END_VAR
// calculate Hour
	arCalculateEnergy_1H[LV01]( lrAccumulator := pmDev.DB07_01_5500.Basic.RealEnergy_IntoLoad);
	arCalculateEnergy_1H[DB_PR1_1]( lrAccumulator := pmDev.DB06_06_5500.Basic.RealEnergy_IntoLoad);
	arCalculateEnergy_1H[DB1]( lrAccumulator := pmDev.DB05_10_5500.Basic.RealEnergy_IntoLoad);
	arCalculateEnergy_1H[DB2]( lrAccumulator := pmDev.DB04_06_5500.Basic.RealEnergy_IntoLoad);
	arCalculateEnergy_1H[DB3]( lrAccumulator := pmDev.DB04_04_5500.Basic.RealEnergy_IntoLoad);
	arCalculateEnergy_1H[DB4]( lrAccumulator := pmDev.DB04_02_5500.Basic.RealEnergy_IntoLoad);
	arCalculateEnergy_1H[DB1_1]( lrAccumulator := pmDev.DB05_09_5350.Basic.RealEnergy_IntoLoad);
	arCalculateEnergy_1H[DB2_1]( lrAccumulator := pmDev.DB04_05_5350.Basic.RealEnergy_IntoLoad);
	arCalculateEnergy_1H[DB3_1]( lrAccumulator := pmDev.DB04_03_5350.Basic.RealEnergy_IntoLoad);
	arCalculateEnergy_1H[DB4_1]( lrAccumulator := pmDev.DB04_01_5350.Basic.RealEnergy_IntoLoad);
	arCalculateEnergy_1H[DB5]( lrAccumulator := pmDev.DB03_04_5500.Basic.RealEnergy_IntoLoad);
	arCalculateEnergy_1H[DB6]( lrAccumulator := pmDev.DB03_06_5500.Basic.RealEnergy_IntoLoad);
	arCalculateEnergy_1H[DB7]( lrAccumulator := pmDev.DB03_02_5500.Basic.RealEnergy_IntoLoad);
	arCalculateEnergy_1H[DB_MR]( lrAccumulator := pmDev.DB06_11_5500.Basic.RealEnergy_IntoLoad);
	arCalculateEnergy_1H[DB5_1]( lrAccumulator := pmDev.DB03_03_5350.Basic.RealEnergy_IntoLoad);
	arCalculateEnergy_1H[DB6_1]( lrAccumulator := pmDev.DB03_05_5350.Basic.RealEnergy_IntoLoad);
	arCalculateEnergy_1H[DB7_1]( lrAccumulator := pmDev.DB03_01_5350.Basic.RealEnergy_IntoLoad);
	arCalculateEnergy_1H[LV02]( lrAccumulator := pmDev.DB07_02_5500.Basic.RealEnergy_IntoLoad);
	arCalculateEnergy_1H[DB_PR1_2]( lrAccumulator := pmDev.DB06_05_5500.Basic.RealEnergy_IntoLoad);
	arCalculateEnergy_1H[DB_AIRCOMP]( lrAccumulator := pmDev.DB07_03_5500.Basic.RealEnergy_IntoLoad);
	arCalculateEnergy_1H[DB_AHU]( lrAccumulator := pmDev.DB06_07_5500.Basic.RealEnergy_IntoLoad);
	arCalculateEnergy_1H[DB8]( lrAccumulator := pmDev.DB05_04_5500.Basic.RealEnergy_IntoLoad);
	arCalculateEnergy_1H[DB9]( lrAccumulator := pmDev.DB05_06_5500.Basic.RealEnergy_IntoLoad);
	arCalculateEnergy_1H[DB10]( lrAccumulator := pmDev.DB05_08_5500.Basic.RealEnergy_IntoLoad);
	arCalculateEnergy_1H[DB8_1]( lrAccumulator := pmDev.DB05_03_5350.Basic.RealEnergy_IntoLoad);
	arCalculateEnergy_1H[DB9_1]( lrAccumulator := pmDev.DB05_05_5350.Basic.RealEnergy_IntoLoad);
	arCalculateEnergy_1H[DB10_1]( lrAccumulator := pmDev.DB05_07_5350.Basic.RealEnergy_IntoLoad);
	arCalculateEnergy_1H[A1]( lrAccumulator := pmDev.DB07_06_5350.Basic.RealEnergy_IntoLoad);
	arCalculateEnergy_1H[A2]( lrAccumulator := pmDev.DB07_07_5350.Basic.RealEnergy_IntoLoad);
	arCalculateEnergy_1H[A3]( lrAccumulator := pmDev.DB07_08_5350.Basic.RealEnergy_IntoLoad);
	arCalculateEnergy_1H[A4]( lrAccumulator := pmDev.DB07_09_5350.Basic.RealEnergy_IntoLoad);
	arCalculateEnergy_1H[A5]( lrAccumulator := pmDev.DB07_10_5350.Basic.RealEnergy_IntoLoad);
	arCalculateEnergy_1H[LP_PR1A]( lrAccumulator := pmDev.DB05_01_5350.Basic.RealEnergy_IntoLoad);
	arCalculateEnergy_1H[LP_PR1B]( lrAccumulator := pmDev.DB05_02_5350.Basic.RealEnergy_IntoLoad);
	arCalculateEnergy_1H[LP_PR2A]( lrAccumulator := pmDev.DB05_22_5350.Basic.RealEnergy_IntoLoad);
	arCalculateEnergy_1H[LP_PR2B]( lrAccumulator := pmDev.DB05_21_5350.Basic.RealEnergy_IntoLoad);
	arCalculateEnergy_1H[LP_PR3A]( lrAccumulator := pmDev.DB03_08_5350.Basic.RealEnergy_IntoLoad);
	arCalculateEnergy_1H[DB_WH]( lrAccumulator := pmDev.DB01_18_5500.Basic.RealEnergy_IntoLoad);
	arCalculateEnergy_1H[LP_PR3B]( lrAccumulator := pmDev.DB03_07_5350.Basic.RealEnergy_IntoLoad);
	arCalculateEnergy_1H[LP_PR4A]( lrAccumulator := pmDev.DB04_08_5350.Basic.RealEnergy_IntoLoad);
	arCalculateEnergy_1H[LP_PR4B]( lrAccumulator := pmDev.DB04_07_5350.Basic.RealEnergy_IntoLoad);
	arCalculateEnergy_1H[LP_BM]( lrAccumulator := pmDev.DB01_20_5500.Basic.RealEnergy_IntoLoad);
	arCalculateEnergy_1H[DB_BM]( lrAccumulator := pmDev.DB01_22_5500.Basic.RealEnergy_IntoLoad);
	arCalculateEnergy_1H[LV03]( lrAccumulator := pmDev.DB06_04_5500.Basic.RealEnergy_IntoLoad);
	arCalculateEnergy_1H[DB_MVAC1]( lrAccumulator := pmDev.DB07_05_5500.Basic.RealEnergy_IntoLoad);
	arCalculateEnergy_1H[DB_MVAC2]( lrAccumulator := pmDev.DB07_04_5500.Basic.RealEnergy_IntoLoad);
	arCalculateEnergy_1H[DB_OFF2]( lrAccumulator := pmDev.DB06_38_5500.Basic.RealEnergy_IntoLoad);
	arCalculateEnergy_1H[LP_EL1]( lrAccumulator := pmDev.DB06_03_5500.Basic.RealEnergy_IntoLoad);
	arCalculateEnergy_1H[LP_EL2]( lrAccumulator := pmDev.DB06_01_5500.Basic.RealEnergy_IntoLoad);
	arCalculateEnergy_1H[DB_OFF1]( lrAccumulator := pmDev.DB06_08_5500.Basic.RealEnergy_IntoLoad);
	arCalculateEnergy_1H[DB_KIT]( lrAccumulator := pmDev.DB06_33_5500.Basic.RealEnergy_IntoLoad);
	arCalculateEnergy_1H[LP_WH2]( lrAccumulator := pmDev.DB01_12_5350.Basic.RealEnergy_IntoLoad);
	arCalculateEnergy_1H[LP_WH1]( lrAccumulator := pmDev.DB01_11_5500.Basic.RealEnergy_IntoLoad);
	arCalculateEnergy_1H[CH4]( lrAccumulator := pmDev.DB07_11_5350.Basic.RealEnergy_IntoLoad);
	arCalculateEnergy_1H[CH5]( lrAccumulator := pmDev.DB07_12_5350.Basic.RealEnergy_IntoLoad);
	arCalculateEnergy_1H[CH6]( lrAccumulator := pmDev.DB07_13_5350.Basic.RealEnergy_IntoLoad);
	arCalculateEnergy_1H[LV04]( lrAccumulator := pmDev.DB06_02_5500.Basic.RealEnergy_IntoLoad);
	arCalculateEnergy_1H[DB_PR2]( lrAccumulator := pmDev.DB01_07_5500.Basic.RealEnergy_IntoLoad);
	arCalculateEnergy_1H[DB11]( lrAccumulator := pmDev.DB01_04_5500.Basic.RealEnergy_IntoLoad);
	arCalculateEnergy_1H[DB12]( lrAccumulator := pmDev.DB01_01_5500.Basic.RealEnergy_IntoLoad);
	arCalculateEnergy_1H[DB13]( lrAccumulator := pmDev.DB02_02_5500.Basic.RealEnergy_IntoLoad);
	arCalculateEnergy_1H[DB14]( lrAccumulator := pmDev.DB02_06_5500.Basic.RealEnergy_IntoLoad);
	arCalculateEnergy_1H[DB11_1]( lrAccumulator := pmDev.DB01_03_5350.Basic.RealEnergy_IntoLoad);
	arCalculateEnergy_1H[DB12_1]( lrAccumulator := pmDev.DB01_02_5350.Basic.RealEnergy_IntoLoad);
	arCalculateEnergy_1H[DB13_1]( lrAccumulator := pmDev.DB02_01_5350.Basic.RealEnergy_IntoLoad);
	arCalculateEnergy_1H[DB14_1]( lrAccumulator := pmDev.DB02_05_5350.Basic.RealEnergy_IntoLoad);
	arCalculateEnergy_1H[DB15]( lrAccumulator := pmDev.DB02_04_5500.Basic.RealEnergy_IntoLoad);
	arCalculateEnergy_1H[DB15_1]( lrAccumulator := pmDev.DB02_03_5350.Basic.RealEnergy_IntoLoad);
	arCalculateEnergy_1H[LP_PR5A]( lrAccumulator := pmDev.DB02_08_5350.Basic.RealEnergy_IntoLoad);
	arCalculateEnergy_1H[LP_PR5B]( lrAccumulator := pmDev.DB02_07_5350.Basic.RealEnergy_IntoLoad);
	arCalculateEnergy_1H[LP_PR6A]( lrAccumulator := pmDev.DB01_06_5350.Basic.RealEnergy_IntoLoad);
	arCalculateEnergy_1H[LP_PR6B]( lrAccumulator := pmDev.DB01_05_5350.Basic.RealEnergy_IntoLoad);
	arCalculateEnergy_1H[DB1_2]( lrAccumulator := pmDev.PowerMeter_DB1_2.Basic.RealEnergy_IntoLoad);
	arCalculateEnergy_1H[DB2_2]( lrAccumulator := pmDev.PowerMeter_DB2_2.Basic.RealEnergy_IntoLoad);
	arCalculateEnergy_1H[DB3_2]( lrAccumulator := pmDev.PowerMeter_DB3_2.Basic.RealEnergy_IntoLoad);
	arCalculateEnergy_1H[DB4_2]( lrAccumulator := pmDev.PowerMeter_DB4_2.Basic.RealEnergy_IntoLoad);
	arCalculateEnergy_1H[DB5_2]( lrAccumulator := pmDev.PowerMeter_DB5_2.Basic.RealEnergy_IntoLoad);
	arCalculateEnergy_1H[DB6_2]( lrAccumulator := pmDev.PowerMeter_DB6_2.Basic.RealEnergy_IntoLoad);
	arCalculateEnergy_1H[DB7_2]( lrAccumulator := pmDev.PowerMeter_DB7_2.Basic.RealEnergy_IntoLoad);
	arCalculateEnergy_1H[DB8_2]( lrAccumulator := pmDev.PowerMeter_DB8_2.Basic.RealEnergy_IntoLoad);
	arCalculateEnergy_1H[DB9_2]( lrAccumulator := pmDev.PowerMeter_DB9_2.Basic.RealEnergy_IntoLoad);
	arCalculateEnergy_1H[DB10_2]( lrAccumulator := pmDev.PowerMeter_DB10_2.Basic.RealEnergy_IntoLoad);
	arCalculateEnergy_1H[DB11_2]( lrAccumulator := pmDev.PowerMeter_DB11_2.Basic.RealEnergy_IntoLoad);
	arCalculateEnergy_1H[DB12_2]( lrAccumulator := pmDev.PowerMeter_DB12_2.Basic.RealEnergy_IntoLoad);
	arCalculateEnergy_1H[DB13_2]( lrAccumulator := pmDev.PowerMeter_DB13_2.Basic.RealEnergy_IntoLoad);
	arCalculateEnergy_1H[DB14_2]( lrAccumulator := pmDev.PowerMeter_DB14_2.Basic.RealEnergy_IntoLoad);
	arCalculateEnergy_1H[DB15_2]( lrAccumulator := pmDev.PowerMeter_DB15_2.Basic.RealEnergy_IntoLoad);
// calculate Day
	arCalculateEnergy_1D[LV01]( lrAccumulator := pmDev.DB07_01_5500.Basic.RealEnergy_IntoLoad);
	arCalculateEnergy_1D[DB_PR1_1]( lrAccumulator := pmDev.DB06_06_5500.Basic.RealEnergy_IntoLoad);
	arCalculateEnergy_1D[DB1]( lrAccumulator := pmDev.DB05_10_5500.Basic.RealEnergy_IntoLoad);
	arCalculateEnergy_1D[DB2]( lrAccumulator := pmDev.DB04_06_5500.Basic.RealEnergy_IntoLoad);
	arCalculateEnergy_1D[DB3]( lrAccumulator := pmDev.DB04_04_5500.Basic.RealEnergy_IntoLoad);
	arCalculateEnergy_1D[DB4]( lrAccumulator := pmDev.DB04_02_5500.Basic.RealEnergy_IntoLoad);
	arCalculateEnergy_1D[DB1_1]( lrAccumulator := pmDev.DB05_09_5350.Basic.RealEnergy_IntoLoad);
	arCalculateEnergy_1D[DB2_1]( lrAccumulator := pmDev.DB04_05_5350.Basic.RealEnergy_IntoLoad);
	arCalculateEnergy_1D[DB3_1]( lrAccumulator := pmDev.DB04_03_5350.Basic.RealEnergy_IntoLoad);
	arCalculateEnergy_1D[DB4_1]( lrAccumulator := pmDev.DB04_01_5350.Basic.RealEnergy_IntoLoad);
	arCalculateEnergy_1D[DB5]( lrAccumulator := pmDev.DB03_04_5500.Basic.RealEnergy_IntoLoad);
	arCalculateEnergy_1D[DB6]( lrAccumulator := pmDev.DB03_06_5500.Basic.RealEnergy_IntoLoad);
	arCalculateEnergy_1D[DB7]( lrAccumulator := pmDev.DB03_02_5500.Basic.RealEnergy_IntoLoad);
	arCalculateEnergy_1D[DB_MR]( lrAccumulator := pmDev.DB06_11_5500.Basic.RealEnergy_IntoLoad);
	arCalculateEnergy_1D[DB5_1]( lrAccumulator := pmDev.DB03_03_5350.Basic.RealEnergy_IntoLoad);
	arCalculateEnergy_1D[DB6_1]( lrAccumulator := pmDev.DB03_05_5350.Basic.RealEnergy_IntoLoad);
	arCalculateEnergy_1D[DB7_1]( lrAccumulator := pmDev.DB03_01_5350.Basic.RealEnergy_IntoLoad);
	arCalculateEnergy_1D[LV02]( lrAccumulator := pmDev.DB07_02_5500.Basic.RealEnergy_IntoLoad);
	arCalculateEnergy_1D[DB_PR1_2]( lrAccumulator := pmDev.DB06_05_5500.Basic.RealEnergy_IntoLoad);
	arCalculateEnergy_1D[DB_AIRCOMP]( lrAccumulator := pmDev.DB07_03_5500.Basic.RealEnergy_IntoLoad);
	arCalculateEnergy_1D[DB_AHU]( lrAccumulator := pmDev.DB06_07_5500.Basic.RealEnergy_IntoLoad);
	arCalculateEnergy_1D[DB8]( lrAccumulator := pmDev.DB05_04_5500.Basic.RealEnergy_IntoLoad);
	arCalculateEnergy_1D[DB9]( lrAccumulator := pmDev.DB05_06_5500.Basic.RealEnergy_IntoLoad);
	arCalculateEnergy_1D[DB10]( lrAccumulator := pmDev.DB05_08_5500.Basic.RealEnergy_IntoLoad);
	arCalculateEnergy_1D[DB8_1]( lrAccumulator := pmDev.DB05_03_5350.Basic.RealEnergy_IntoLoad);
	arCalculateEnergy_1D[DB9_1]( lrAccumulator := pmDev.DB05_05_5350.Basic.RealEnergy_IntoLoad);
	arCalculateEnergy_1D[DB10_1]( lrAccumulator := pmDev.DB05_07_5350.Basic.RealEnergy_IntoLoad);
	arCalculateEnergy_1D[A1]( lrAccumulator := pmDev.DB07_06_5350.Basic.RealEnergy_IntoLoad);
	arCalculateEnergy_1D[A2]( lrAccumulator := pmDev.DB07_07_5350.Basic.RealEnergy_IntoLoad);
	arCalculateEnergy_1D[A3]( lrAccumulator := pmDev.DB07_08_5350.Basic.RealEnergy_IntoLoad);
	arCalculateEnergy_1D[A4]( lrAccumulator := pmDev.DB07_09_5350.Basic.RealEnergy_IntoLoad);
	arCalculateEnergy_1D[A5]( lrAccumulator := pmDev.DB07_10_5350.Basic.RealEnergy_IntoLoad);
	arCalculateEnergy_1D[LP_PR1A]( lrAccumulator := pmDev.DB05_01_5350.Basic.RealEnergy_IntoLoad);
	arCalculateEnergy_1D[LP_PR1B]( lrAccumulator := pmDev.DB05_02_5350.Basic.RealEnergy_IntoLoad);
	arCalculateEnergy_1D[LP_PR2A]( lrAccumulator := pmDev.DB05_22_5350.Basic.RealEnergy_IntoLoad);
	arCalculateEnergy_1D[LP_PR2B]( lrAccumulator := pmDev.DB05_21_5350.Basic.RealEnergy_IntoLoad);
	arCalculateEnergy_1D[LP_PR3A]( lrAccumulator := pmDev.DB03_08_5350.Basic.RealEnergy_IntoLoad);
	arCalculateEnergy_1D[DB_WH]( lrAccumulator := pmDev.DB01_18_5500.Basic.RealEnergy_IntoLoad);
	arCalculateEnergy_1D[LP_PR3B]( lrAccumulator := pmDev.DB03_07_5350.Basic.RealEnergy_IntoLoad);
	arCalculateEnergy_1D[LP_PR4A]( lrAccumulator := pmDev.DB04_08_5350.Basic.RealEnergy_IntoLoad);
	arCalculateEnergy_1D[LP_PR4B]( lrAccumulator := pmDev.DB04_07_5350.Basic.RealEnergy_IntoLoad);
	arCalculateEnergy_1D[LP_BM]( lrAccumulator := pmDev.DB01_20_5500.Basic.RealEnergy_IntoLoad);
	arCalculateEnergy_1D[DB_BM]( lrAccumulator := pmDev.DB01_22_5500.Basic.RealEnergy_IntoLoad);
	arCalculateEnergy_1D[LV03]( lrAccumulator := pmDev.DB06_04_5500.Basic.RealEnergy_IntoLoad);
	arCalculateEnergy_1D[DB_MVAC1]( lrAccumulator := pmDev.DB07_05_5500.Basic.RealEnergy_IntoLoad);
	arCalculateEnergy_1D[DB_MVAC2]( lrAccumulator := pmDev.DB07_04_5500.Basic.RealEnergy_IntoLoad);
	arCalculateEnergy_1D[DB_OFF2]( lrAccumulator := pmDev.DB06_38_5500.Basic.RealEnergy_IntoLoad);
	arCalculateEnergy_1D[LP_EL1]( lrAccumulator := pmDev.DB06_03_5500.Basic.RealEnergy_IntoLoad);
	arCalculateEnergy_1D[LP_EL2]( lrAccumulator := pmDev.DB06_01_5500.Basic.RealEnergy_IntoLoad);
	arCalculateEnergy_1D[DB_OFF1]( lrAccumulator := pmDev.DB06_08_5500.Basic.RealEnergy_IntoLoad);
	arCalculateEnergy_1D[DB_KIT]( lrAccumulator := pmDev.DB06_33_5500.Basic.RealEnergy_IntoLoad);
	arCalculateEnergy_1D[LP_WH2]( lrAccumulator := pmDev.DB01_12_5350.Basic.RealEnergy_IntoLoad);
	arCalculateEnergy_1D[LP_WH1]( lrAccumulator := pmDev.DB01_11_5500.Basic.RealEnergy_IntoLoad);
	arCalculateEnergy_1D[CH4]( lrAccumulator := pmDev.DB07_11_5350.Basic.RealEnergy_IntoLoad);
	arCalculateEnergy_1D[CH5]( lrAccumulator := pmDev.DB07_12_5350.Basic.RealEnergy_IntoLoad);
	arCalculateEnergy_1D[CH6]( lrAccumulator := pmDev.DB07_13_5350.Basic.RealEnergy_IntoLoad);
	arCalculateEnergy_1D[LV04]( lrAccumulator := pmDev.DB06_02_5500.Basic.RealEnergy_IntoLoad);
	arCalculateEnergy_1D[DB_PR2]( lrAccumulator := pmDev.DB01_07_5500.Basic.RealEnergy_IntoLoad);
	arCalculateEnergy_1D[DB11]( lrAccumulator := pmDev.DB01_04_5500.Basic.RealEnergy_IntoLoad);
	arCalculateEnergy_1D[DB12]( lrAccumulator := pmDev.DB01_01_5500.Basic.RealEnergy_IntoLoad);
	arCalculateEnergy_1D[DB13]( lrAccumulator := pmDev.DB02_02_5500.Basic.RealEnergy_IntoLoad);
	arCalculateEnergy_1D[DB14]( lrAccumulator := pmDev.DB02_06_5500.Basic.RealEnergy_IntoLoad);
	arCalculateEnergy_1D[DB11_1]( lrAccumulator := pmDev.DB01_03_5350.Basic.RealEnergy_IntoLoad);
	arCalculateEnergy_1D[DB12_1]( lrAccumulator := pmDev.DB01_02_5350.Basic.RealEnergy_IntoLoad);
	arCalculateEnergy_1D[DB13_1]( lrAccumulator := pmDev.DB02_01_5350.Basic.RealEnergy_IntoLoad);
	arCalculateEnergy_1D[DB14_1]( lrAccumulator := pmDev.DB02_05_5350.Basic.RealEnergy_IntoLoad);
	arCalculateEnergy_1D[DB15]( lrAccumulator := pmDev.DB02_04_5500.Basic.RealEnergy_IntoLoad);
	arCalculateEnergy_1D[DB15_1]( lrAccumulator := pmDev.DB02_03_5350.Basic.RealEnergy_IntoLoad);
	arCalculateEnergy_1D[LP_PR5A]( lrAccumulator := pmDev.DB02_08_5350.Basic.RealEnergy_IntoLoad);
	arCalculateEnergy_1D[LP_PR5B]( lrAccumulator := pmDev.DB02_07_5350.Basic.RealEnergy_IntoLoad);
	arCalculateEnergy_1D[LP_PR6A]( lrAccumulator := pmDev.DB01_06_5350.Basic.RealEnergy_IntoLoad);
	arCalculateEnergy_1D[LP_PR6B]( lrAccumulator := pmDev.DB01_05_5350.Basic.RealEnergy_IntoLoad);
	arCalculateEnergy_1D[DB1_2]( lrAccumulator := pmDev.PowerMeter_DB1_2.Basic.RealEnergy_IntoLoad);
	arCalculateEnergy_1D[DB2_2]( lrAccumulator := pmDev.PowerMeter_DB2_2.Basic.RealEnergy_IntoLoad);
	arCalculateEnergy_1D[DB3_2]( lrAccumulator := pmDev.PowerMeter_DB3_2.Basic.RealEnergy_IntoLoad);
	arCalculateEnergy_1D[DB4_2]( lrAccumulator := pmDev.PowerMeter_DB4_2.Basic.RealEnergy_IntoLoad);
	arCalculateEnergy_1D[DB5_2]( lrAccumulator := pmDev.PowerMeter_DB5_2.Basic.RealEnergy_IntoLoad);
	arCalculateEnergy_1D[DB6_2]( lrAccumulator := pmDev.PowerMeter_DB6_2.Basic.RealEnergy_IntoLoad);
	arCalculateEnergy_1D[DB7_2]( lrAccumulator := pmDev.PowerMeter_DB7_2.Basic.RealEnergy_IntoLoad);
	arCalculateEnergy_1D[DB8_2]( lrAccumulator := pmDev.PowerMeter_DB8_2.Basic.RealEnergy_IntoLoad);
	arCalculateEnergy_1D[DB9_2]( lrAccumulator := pmDev.PowerMeter_DB9_2.Basic.RealEnergy_IntoLoad);
	arCalculateEnergy_1D[DB10_2]( lrAccumulator := pmDev.PowerMeter_DB10_2.Basic.RealEnergy_IntoLoad);
	arCalculateEnergy_1D[DB11_2]( lrAccumulator := pmDev.PowerMeter_DB11_2.Basic.RealEnergy_IntoLoad);
	arCalculateEnergy_1D[DB12_2]( lrAccumulator := pmDev.PowerMeter_DB12_2.Basic.RealEnergy_IntoLoad);
	arCalculateEnergy_1D[DB13_2]( lrAccumulator := pmDev.PowerMeter_DB13_2.Basic.RealEnergy_IntoLoad);
	arCalculateEnergy_1D[DB14_2]( lrAccumulator := pmDev.PowerMeter_DB14_2.Basic.RealEnergy_IntoLoad);
	arCalculateEnergy_1D[DB15_2]( lrAccumulator := pmDev.PowerMeter_DB15_2.Basic.RealEnergy_IntoLoad);
//FIFO Hour
	// // Check NEw Hour ( in the last Meter => it's mean all the calculate in 1 hour is updated)	
	IF arCalculateEnergy_1H[pmDev.numAllMeter-1].bNewPeriodAlarm THEN
		FIFOEnergyTimestruct_1H.MR_AddValue( Value := arCalculateEnergy_1H[pmDev.numAllMeter-1].previousTimestampOut);
		FOR iLoop := 0 TO pmDev.numAllMeter-1 DO
			arFIFOEnergy_1H[iLoop].MR_AddValue( Value := arCalculateEnergy_1H[iLoop].accumulatedValueOut);
			arCalculateEnergy_1H[iLoop].MR_Acknowledge();
		END_FOR
	END_IF	
// Check NEw Day ( in the last Meter => it's mean all the calculate in 1 day is updated)	
	IF arCalculateEnergy_1D[pmDev.numAllMeter-1].bNewPeriodAlarm THEN
		FIFOEnergyTimestruct_1D.MR_AddValue(  Value := arCalculateEnergy_1H[pmDev.numAllMeter-1].previousTimestampOut);
		FOR iLoop := 0 TO pmDev.numAllMeter-1 DO
			// round number before go to the FIFO
			arFIFOEnergy_1D[iLoop].MR_AddValue(
				Value := F_RoundLrealEx( 
					lrIn := arCalculateEnergy_1D[iLoop].accumulatedValueOut,
					iPrecision := 0)
			);
			// Ack The Calculate
			arCalculateEnergy_1D[iloop].MR_Acknowledge();
		END_FOR

	END_IF
	
CASE eStateReport OF
	STATE_REPORT_WAIT:
		// Check the last one FIFO[-1] hour if have data => request report to Aveva.
			IF arFIFOEnergy_1H[pmDev.numAllMeter-1].DataReady  THEN
				eStateReport := STATE_REPORT_ENERGY_HOUR_REQUEST;
		// Check the last one FIFO[-1] hour if have data => request report to Aveva.
			ELSIF arFIFOEnergy_1D[pmDev.numAllMeter-1].DataReady  THEN
				eStateReport := STATE_REPORT_ENERGY_DAY_REQUEST;
			END_IF;
			
	STATE_REPORT_ENERGY_HOUR_REQUEST:
		sDateAndTimeReportAveva := TimeStruct_To_sTimeAveva(timestruct := FIFOEnergyTimestruct_1H.OldestData, typeFormat := 5 );
		sMsReportAveva			:= WORD_TO_STRING ( FIFOEnergyTimestruct_1H.OldestData.wMilliseconds);
		
		fbMachineLogger.MR_AddLogs( sLogMessage :=  CONCAT('REPORT_ENERGY_HOUR_REQUEST  ', sDateAndTimeReportAveva  ));
		eStateReport := STATE_REPORT_ENERGY_HOUR_ACTIVE_REQUEST;
	
	STATE_REPORT_ENERGY_HOUR_ACTIVE_REQUEST	:
		tonPrepareValue( IN := TRUE,
							PT := tTimePrepareValue);
		IF tonPrepareValue.Q THEN
			tonPrepareValue( IN := FALSE);
			bEnergyReportHourEvent := TRUE;
			eStateReport := STATE_REPORT_ENERGY_HOUR_WAIT_ACK;
		END_IF
	
	STATE_REPORT_ENERGY_HOUR_WAIT_ACK:
		IF bEnergyReportHourEvent = FALSE THEN
			FOR iLoop := 0 TO pmDev.numAllMeter-1 DO
				arFIFOEnergy_1H[iLoop].MR_AckGetValue();
			END_FOR
			FIFOEnergyTimestruct_1H.MR_AckGetValue();
			fbMachineLogger.MR_AddLogs( sLogMessage :=  'REPORT_ENERGY_HOUR_ACKed  ');
			eStateReport := STATE_REPORT_WAIT;
		END_IF
				
	STATE_REPORT_ENERGY_DAY_REQUEST:
		CalculateVirtualObject();
		sDateAndTimeReportAveva := TimeStruct_To_sTimeAveva(timestruct := FIFOEnergyTimestruct_1D.OldestData, typeFormat := 5 );
	 	sMsReportAveva			:= WORD_TO_STRING ( FIFOEnergyTimestruct_1D.OldestData.wMilliseconds);
		bEnergyReportDayEvent := TRUE;
		fbMachineLogger.MR_AddLogs( sLogMessage :=  CONCAT('REPORT_ENERGY_DAY_REQUEST  ', sDateAndTimeReportAveva  ));
		eStateReport := STATE_REPORT_ENERGY_DAY_ACTIVE_REQUEST;
		
	STATE_REPORT_ENERGY_DAY_ACTIVE_REQUEST	:
		tonPrepareValue( IN := TRUE,
							PT := tTimePrepareValue);
		IF tonPrepareValue.Q THEN
			tonPrepareValue( IN := FALSE);
			bEnergyReportDayEvent := TRUE;
			eStateReport := STATE_REPORT_ENERGY_DAY_WAIT_ACK;
		END_IF	
		
	STATE_REPORT_ENERGY_DAY_WAIT_ACK:
		IF bEnergyReportDayEvent = FALSE THEN
			FOR iLoop := 0 TO pmDev.numAllMeter-1 DO
				arFIFOEnergy_1D[iLoop].MR_AckGetValue();	
			END_FOR

			FIFOEnergyTimestruct_1D.MR_AckGetValue();
			fbMachineLogger.MR_AddLogs( sLogMessage :=  'REPORT_ENERGY_HOUR_ACKed  ');
			eStateReport := STATE_REPORT_WAIT;
		END_IF
END_CASE
END_METHOD

END_PROGRAM

// ---- POUs/CalAccum/FB_CalCulateAccumulation.TcPOU
FUNCTION_BLOCK FB_CalCulateAccumulation
VAR_INPUT
	lrAccumulator : LREAL  := 0;
	
END_VAR
VAR_OUTPUT
	accumulatedValueOut : LREAL;// value = lrAccumulator(timeNew) - lrAccumulator(timeOld)
	previousTimestampOut	: TIMESTRUCT;// TimeOld
	bNewPeriodAlarm : BOOL;// Remain True in 30s if not be ackNowledge
	
END_VAR
VAR

	
	eCpHour		: E_CompareTime;
	eCpDay 		: E_CompareTime;
	eCpMonth	: E_CompareTime;
	eCpYear		: E_CompareTime;
	eCpMinute	: E_CompareTime;
	eSameTime : E_CompareTime;
	eNewTime : E_CompareTime;
	eRfTimeCompare : REFERENCE TO E_CompareTime;
	sName 		: STRING;
	eState : UINT;
	TonRemainOutput : TON;
	eTimeAccumulate : E_CompareTime;
	bInit : BOOL;
	bReset : BOOL;
	bRequestUpdate_ValueInLastTime: BOOL;
END_VAR

VAR PERSISTENT 
	bUpdatedValueLastHour : BOOL;// reject Power OFF unexpected
	previousTimestamp	: TIMESTRUCT;
	ValueInLastTime : LREAL;
	accumulatedValue : LREAL;
	
	
END_VAR
VAR CONSTANT
	eStateUinitialized : UINT := 0;
	eStateInit : UINT := 10;
	eStateRun : UINT := 20;
	eStateReset : UINT := 100;
	TimeNewPeriodAlarm : TIME := T#30s;
END_VAR



				
CASE eState OF
	eStateUinitialized: // unInitialized
		;// will go to eStateInit if MR_Run is called 
		
	eStateInit: 
		;// will call by MR_Init
		
	eStateRun: //StateRun
		MS_Run();
		
	eStateReset :
		MS_Reset();
	
END_CASE

IF eState > 0 AND bReset THEN
	eState := eStateReset;
END_IF

PROPERTY isInitDone : bool
GET
END_GET
END_PROPERTY

PROPERTY isRuning : bool
GET
isRuning := eState = eStateRun;
END_GET
END_PROPERTY

// if not return true , check the Current time and PreviousTime in fb
METHOD MR_Acknowledge : BOOL
VAR_INPUT
END_VAR
bNewPeriodAlarm := FALSE;
IF eRfTimeCompare = eSameTime THEN
	MR_Acknowledge := TRUE;
END_IF
END_METHOD

METHOD MR_Init : BOOL
VAR_INPUT
END_VAR

IF eState = eStateUinitialized THEN// init;
	bInit := true;
 
	IF MS_Init() THEN
		MR_Init := TRUE;
		eState := eStateRun;
	END_IF


END_IF
END_METHOD

METHOD MR_Reset : BOOL
VAR_INPUT
END_VAR
bReset := TRUE;
IF eState = eStateUinitialized THEN
	MR_Reset := TRUE;
	bReset := false;
END_IF
END_METHOD

METHOD Protected MS_Init : BOOL
VAR_INPUT
END_VAR
CASE eTimeAccumulate OF
	NEW_MINUTE :
		eSameTime := SAME_MINUTE;
		eNewTime := NEW_MINUTE;
		eRfTimeCompare REF= eCpMinute;
		MS_Init := TRUE;
	NEW_HOUR :
		eSameTime := SAME_HOUR;
		eNewTime := NEW_HOUR;
		eRfTimeCompare REF= eCpHour;
		MS_Init := TRUE;
	NEW_DAY	:
		eSameTime := SAME_DAY;
		eNewTime := NEW_DAY;
		eRfTimeCompare REF= eCpDay;
		MS_Init := TRUE;
	NEW_MONTH:
		eSameTime := SAME_MONTH;
		eNewTime := NEW_MONTH;
		eRfTimeCompare REF= eCpMonth;
		MS_Init := TRUE;
	NEW_YEAR:
		eSameTime := SAME_YEAR;
		eNewTime := NEW_YEAR;
		eRfTimeCompare REF= eCpYear;
		MS_Init := true;
END_CASE
END_METHOD

METHOD protected MS_Reset : BOOL
VAR_INPUT
END_VAR
//retainvalue
	
	bUpdatedValueLastHour := FALSE;
	previousTimestamp.wYear := 0;
	previousTimestamp.wMonth := 0;
	previousTimestamp.wDay := 0;
	previousTimestamp.wMinute := 0;
	previousTimestamp.wSecond := 0;
	previousTimestamp.wMilliseconds := 0;
	ValueInLastTime := 0 ;
	accumulatedValue := 0 ;
// out_put
	accumulatedValueOut := 0;
	previousTimestampOut.wYear := 0;
	previousTimestampOut.wMonth := 0;
	previousTimestampOut.wDay := 0;
	previousTimestampOut.wMinute := 0;
	previousTimestampOut.wSecond := 0;
	previousTimestampOut.wMilliseconds := 0;
	bNewPeriodAlarm := false;// Remain True 
	
// 	RETURN TO uninit
	eState := eStateUinitialized;
	eRfTimeCompare REF= 0;
END_METHOD

METHOD Protected MS_Run : BOOL
VAR_INPUT
END_VAR
	CompareTime(	timestruct1 := previousTimestamp,
					timestruct2 := GVL.fbMachineTime.systemTime,
					eCpMinute => eCpMinute, 
					eCpHour => eCpHour,
					eCpDay => eCpDay,
					eCpMonth => eCpMonth,
					ecpYear => eCpYear);

	IF eRfTimeCompare = eNewTime THEN
		// update to output
		accumulatedValueOut := accumulatedValue;
		previousTimestampOut := previousTimestamp;
		bNewPeriodAlarm := TRUE;
		// update the the last hour and time
		bUpdatedValueLastHour := FALSE;
		IF lrAccumulator > 0.1 THEN
			ValueInLastTime := lrAccumulator;
			bRequestUpdate_ValueInLastTime := FALSE;
			// UpdateOK
			bUpdatedValueLastHour := TRUE;
		ELSE
			bRequestUpdate_ValueInLastTime := TRUE;
		END_IF
		ValueInLastTime := lrAccumulator;
		previousTimestamp := GVL.fbMachineTime.systemTime;

	
	ELSIF eRfTimeCompare = eSameTime AND bUpdatedValueLastHour THEN
		IF lrAccumulator > 0.1 THEN // reject the situation that just TURN ON IPC so lrAccumulator = -8888888888888888.444444444444
			accumulatedValue := lrAccumulator - ValueInLastTime;
		END_IF
	ELSIF eRfTimeCompare = eSameTime AND NOT bUpdatedValueLastHour THEN
		ValueInLastTime := lrAccumulator;
		previousTimestamp := GVL.fbMachineTime.systemTime;
	ELSE
		; //invalid time Compare
	

	END_IF
	
TonRemainOutput( IN := bNewPeriodAlarm , PT := TimeNewPeriodAlarm);

IF TonRemainOutput.Q THEN
	bNewPeriodAlarm := false;
END_IF
IF bRequestUpdate_ValueInLastTime THEN
	IF lrAccumulator > 0.1 THEN
		ValueInLastTime := lrAccumulator;
		bRequestUpdate_ValueInLastTime := FALSE;
		// UpdateOK
		bUpdatedValueLastHour := TRUE;
	END_IF
END_IF
END_METHOD

PROPERTY Name : string
GET
Name := sName;
END_GET
SET
sName := Name;
END_SET
END_PROPERTY

// Set TimeAccumulate before call Mr_Init.
//NEW_MINUTE := 5,
//	NEW_HOUR := 10,
//	NEW_DAY	:= 20,
//	NEW_MONTH := 30,
//	NEW_YEAR	:= 32,
PROPERTY TimeAccumulate : E_CompareTime
GET
TimeAccumulate := eTimeAccumulate;
END_GET
SET
eTimeAccumulate := TimeAccumulate;
END_SET
END_PROPERTY

END_FUNCTION_BLOCK

// ---- Function/CompareTime.TcPOU
FUNCTION CompareTime : E_CompareTime
VAR_INPUT
		timestruct1 : TIMESTRUCT;//TIMEPREVIOUS
		timestruct2 : TIMESTRUCT;// TIME NOW
END_VAR
VAR_OUTPUT
	eCpMinute	: E_CompareTime;
	eCpHour		: E_CompareTime;
	eCpDay		: E_CompareTime;
	eCpMonth	: E_CompareTime;
	ecpYear		: E_CompareTime;
END_VAR

IF timestruct1.wYear < timestruct2.wYear THEN
	CompareTime := NEW_YEAR;
	ecpYear := NEW_YEAR;
	eCpMonth := NEW_MONTH;
	eCpDay := NEW_DAY;
	eCpHour := NEW_HOUR;
	eCpMinute := NEW_MINUTE;
ELSIF timestruct1.wYear > timestruct2.wYear THEN
		CompareTime := INVALID_PRE_TIME;
ELSE 
	ecpYear := SAME_YEAR;
	IF timestruct1.wMonth < timestruct2.wMonth THEN
		CompareTime := NEW_MONTH;
		eCpMonth := NEW_MONTH;
		eCpDay := NEW_DAY;
		eCpHour := NEW_HOUR;
		eCpMinute := NEW_MINUTE;
	ELSIF  timestruct1.wMonth > timestruct2.wMonth THEN
			CompareTime := INVALID_PRE_TIME;
	ELSE
		eCpMonth := SAME_MONTH;
		IF timestruct1.wDay < timestruct2.wDay THEN
			CompareTime := NEW_DAY;
			eCpDay := NEW_DAY;
			eCpHour := NEW_HOUR;
			eCpMinute := NEW_MINUTE;
		ELSIF timestruct1.wDay > timestruct2.wDay THEN
			CompareTime := INVALID_PRE_TIME;
		ELSE 
			eCpDay := SAME_DAY;
			IF timestruct1.wHour < timestruct2.wHour THEN
				CompareTime := NEW_HOUR;
				eCpHour := NEW_HOUR;
				eCpMinute := NEW_MINUTE;
			ELSIF timestruct1.wHour > timestruct2.wHour THEN
				CompareTime := INVALID_PRE_TIME; 
			ELSE
				eCpHour := SAME_HOUR;
				IF timestruct1.wMinute < timestruct2.wMinute THEN
					CompareTime := NEW_MINUTE;
					eCpMinute := NEW_MINUTE;
				ELSIF timestruct1.wMinute > timestruct2.wMinute THEN
					CompareTime := INVALID_PRE_TIME; 
				ELSE
					CompareTime := SAME_MINUTE;	
					eCpMinute := SAME_MINUTE;
			END_IF
			END_IF
		END_IF

	END_IF
END_IF

END_FUNCTION

// ---- POUs/FIFO/FB_FIFO_Lreal.TcPOU
FUNCTION_BLOCK FB_FIFO_Lreal EXTENDS FB_Universal_FIFO IMPLEMENTS I_FIFO_Lreal
VAR_INPUT
  
END_VAR

VAR
  
END_VAR

VAR_OUTPUT
	OldestData : LREAL;
END_VAR
VAR PERSISTENT
	Queue : ARRAY[0..MaxQueueSize-1] OF LREAL;  // FIFO queue (size is 100 elements)
END_VAR



//    // Log new data only if LogData is TRUE
//    IF rTrigLogData.Q THEN
//        IF Count < MaxQueueSize THEN
//            Queue[Head] := NewEnergyData;
//            Head := (Head + 1) MOD MaxQueueSize;
//            Count := Count + 1;
//        ELSE
//            // FIFO is full, overwrite old data if needed
//            Tail := (Tail + 1) MOD MaxQueueSize;
//            Queue[Head] := NewEnergyData;
//            Head := (Head + 1) MOD MaxQueueSize;
//            // Tail position is updated
//        END_IF
//        DataReady := TRUE;  // New data is now ready to be processed
     
//    END_IF

    // Retrieve and manage oldest data for processing

// if dataready return true, else return false
METHOD  MR_AckGetValue : BOOL
VAR_INPUT
END_VAR
SUPER^.MR_AckGetValue();
  OldestData := Queue[Tail];
 MR_AckGetValue := true;
END_METHOD

METHOD MR_AddValue : BOOL
VAR_INPUT
		Value : LREAL;
END_VAR
  IF Count < MaxQueueSize THEN
            Queue[Head] := Value;
            Head := (Head + 1) MOD MaxQueueSize;
            Count := Count + 1;
  ELSE
            // FIFO is full, overwrite old data if needed
            Tail := (Tail + 1) MOD MaxQueueSize;
            Queue[Head] := Value;
            Head := (Head + 1) MOD MaxQueueSize;
            // Tail position is updated
			
  END_IF
  
  OldestData := Queue[Tail];
  bDataReady := TRUE; 
  
  
  MR_AddValue := true;
END_METHOD

// need overide to reset oldestValue
METHOD MR_Reset : BOOL
VAR_INPUT
END_VAR
SUPER^.MR_Reset();
OldestData := 0;
MR_Reset := true;
END_METHOD

PROPERTY oOldestValue : Lreal
GET
oOldestValue := OldestData;
END_GET
END_PROPERTY

END_FUNCTION_BLOCK

// ---- POUs/FIFO/FB_Universal_FIFO.TcPOU
FUNCTION_BLOCK ABSTRACT FB_Universal_FIFO IMPLEMENTS I_Universal_FIFO

VAR PERSISTENT    
	//Queue : ARRAY[0..MaxQueueSize-1] OF REAL;  // FIFO queue (size is 100 elements)
    Head : UINT := 0;  // Points to the next position to store data
    Tail : UINT := 0;  // Points to the oldest data position
    Count : UINT := 0;  // Number of elements currently in the FIFO
	bDataReady : BOOL; 
	eState : UINT;
END_VAR

VAR CONSTANT
	MaxQueueSize : UINT := 255;  // Number of elements in the FIFO queue

END_VAR

VAR_OUTPUT

   
END_VAR

PROPERTY DataReady : BOOL
GET
DataReady := bDataReady;
END_GET
END_PROPERTY

PROPERTY HeadIndex : UINT
GET
HeadIndex := Head;
END_GET
END_PROPERTY

PROPERTY IsEmpty : bool
GET
IF Count = 0 THEN
	IsEmpty := TRUE;
ELSE
	IsEmpty := false;
END_IF
END_GET
END_PROPERTY

PROPERTY IsFull : bool
GET
IF count = MaxQueueSize THEN
	IsFull := TRUE;
ELSE 
	IsFull := FALSE;
END_IF
END_GET
END_PROPERTY

// if dataready return true, else return false// need overiding a part
METHOD MR_AckGetValue : BOOL
VAR_INPUT
END_VAR
IF bDataReady THEN
      
            // Data has been processed, so move to the next item in the queue
            Tail := (Tail + 1) MOD MaxQueueSize;
            Count := Count - 1;
            IF Count = 0 THEN
                bDataReady := FALSE;  // No more data to process
            END_IF
        
            // Data is still ready to be processed
        
    MR_AckGetValue := TRUE;   
ELSE 
	MR_AckGetValue := FALSE;
END_IF
// set oldest value in child fb here
// OldestData :=   Queue[Tail];
/////
END_METHOD

// need overide to reset oldestValue
METHOD MR_Reset : BOOL
VAR_INPUT
END_VAR
     Head := 0;
     Tail := 0;
     Count := 0;
	 bDataReady := FALSE;
	 MR_Reset := TRUE;
END_METHOD

PROPERTY TailIndex : Uint
GET
TailIndex := Tail;
END_GET
END_PROPERTY

END_FUNCTION_BLOCK

// ---- Function/TimeStruct_To_sTimeAveva.TcPOU
FUNCTION TimeStruct_To_sTimeAveva : STRING// convert TIMESTRUCT TO MONTH/DAY/YEAR HOUR:MINUTE: SECOND ( FORMAT 'MM/DD/YYYY HH:MM:SS' )
VAR_INPUT
	timestruct 	: TIMESTRUCT;
	typeFormat	: UINT := 0; (* 	0: 'MM/DD/YYYY HH:MM:SS'
									1: 'MMDDYYYY'
									2: 'YYYYMMDD'
									3: 'DDMMYYYY'
									4: 'YYYY-MM-DD HH:MM:SS' 
									5: 'YYYY-MM-DD HH:MM:SS.XXX'
													*)
	
END_VAR
VAR
	sYear : STRING;
	sMonth : STRING;
	sDay : STRING;
	sHour : STRING;
	sMinute : STRING;
	sSecond : STRING;
	sMilisecond	: STRING;
	concate1 : STRING;
	
END_VAR

	sYear := WORD_TO_STRING(timestruct.wYear);
	sMonth := WORD_TO_STRING(timestruct.wMonth);
	sDay 	:= WORD_TO_STRING(timestruct.wDay);
	
	sHour := WORD_TO_STRING(timestruct.wHour);
	sMinute := WORD_TO_STRING(timestruct.wMinute);
	sSecond 	:= WORD_TO_STRING(timestruct.wSecond);
	sMilisecond := WORD_TO_STRING(timestruct.wMilliseconds);
	
	IF timestruct.wMonth <10 THEN
		sMonth := CONCAT('0', smonth);
	END_IF
	
	IF timestruct.wDay <10 THEN
		sDay := CONCAT('0', sday);
	END_IF
	
	IF timestruct.wHour <10 THEN
		sHour := CONCAT('0', shour);
	END_IF
	IF timestruct.wSecond <10 THEN
		ssecond := CONCAT('0', ssecond);
	END_IF
	IF timestruct.wMinute <10 THEN
		sMinute := CONCAT('0', sminute);
	END_IF
	
	IF timestruct.wMilliseconds < 10  THEN
		sMilisecond :=  CONCAT('00', sMilisecond);
	ELSIF timestruct.wMilliseconds < 100 THEN
		sMilisecond :=  CONCAT('0', sMilisecond);
	END_IF
	
CASE typeFormat OF
	0://0: 'MM/DD/YYYY HH:MM:SS'
		concate1 := CONCAT( smonth, '/');
		concate1 := CONCAT( concate1, sDay);
		concate1 := CONCAT( concate1, '/');
		concate1 := CONCAT( concate1, sYear);
		concate1 := CONCAT( concate1, ' ');
		concate1 := CONCAT( concate1, shour);
		concate1 := CONCAT( concate1, ':');
		concate1 := CONCAT( concate1, sminute);
		concate1 := CONCAT( concate1, ':');
		concate1 := CONCAT( concate1, ssecond);
	
	1: //1: 'MMDDYYYY'
		concate1 := CONCAT( smonth, sDay);
		concate1 := CONCAT( concate1, sYear);
		
	2: 	//2: 'YYYYMMDD'
		concate1 := CONCAT( syear, smonth);
		concate1 := CONCAT( concate1, sday);	
		
	3: 	//3: 'DDMMYYYY'
		concate1 := CONCAT( sday, smonth);
		concate1 := CONCAT( concate1, syear);	
	4: //'YYYY-MM-DD HH:MM:SS' 
		concate1 := CONCAT( syear, '-');//YYYY-
		concate1 := CONCAT ( concate1, smonth);//YYYY-MM
		concate1 := CONCAT( concate1, '-');//YYYY-MM-
		concate1 := CONCAT( concate1, SDAY);//YYYY-MM-DD
		concate1 := CONCAT( concate1, ' ');//'YYYY-MM-DD '
		concate1 := CONCAT( concate1, shour);//'YYYY-MM-DD HH
		concate1 := CONCAT( concate1, ':');//'YYYY-MM-DD HH:
		concate1 := CONCAT( concate1, sminute);//'YYYY-MM-DD HH:MM
		concate1 := CONCAT( concate1, ':');//'YYYY-MM-DD HH:MM:
		concate1 := CONCAT( concate1, ssecond);//'YYYY-MM-DD HH:MM:SS
	5: (*need addition code*)
		concate1 := CONCAT( syear, '-');//YYYY-
		concate1 := CONCAT ( concate1, smonth);//YYYY-MM
		concate1 := CONCAT( concate1, '-');//YYYY-MM-
		concate1 := CONCAT( concate1, SDAY);//YYYY-MM-DD
		concate1 := CONCAT( concate1, ' ');//'YYYY-MM-DD '
		concate1 := CONCAT( concate1, shour);//'YYYY-MM-DD HH
		concate1 := CONCAT( concate1, ':');//'YYYY-MM-DD HH:
		concate1 := CONCAT( concate1, sminute);//'YYYY-MM-DD HH:MM
		concate1 := CONCAT( concate1, ':');//'YYYY-MM-DD HH:MM:
		concate1 := CONCAT( concate1, ssecond);//'YYYY-MM-DD HH:MM:SS
		concate1 := CONCAT( concate1, '.');//'YYYY-MM-DD HH:MM:SS.
		concate1 := CONCAT( concate1, sMilisecond); ////'YYYY-MM-DD HH:MM:SS.xxx
		
	ELSE
		concate1 := '';
END_CASE

TimeStruct_To_sTimeAveva := concate1;

END_FUNCTION

// ---- Function/FgenerateRandom.TcPOU
FUNCTION FgenerateRandom : Lreal // := rawValue + rawValue*percent* random
VAR_INPUT
	percent : LREAL ;// percent of vabration random +percent
	rawValue : LREAL;
	ValueDrandGenerate : LREAL;
END_VAR
VAR_OUTPUT
	
END_VAR
VAR
	
	
END_VAR

FgenerateRandom := rawValue + rawValue * percent * ValueDrandGenerate;

END_FUNCTION

// ---- TEST/FB_PmSimulate.TcPOU
FUNCTION_BLOCK FB_PmSimulate
VAR
	PM : REFERENCE TO ST_PowerMeter;	
END_VAR 

VAR
	sName : STRING;
	Param : REFERENCE TO ST_PMGeneral;
	bFirstCycle : BOOL := TRUE;
	estate : E_PM_Simulate;
	tonReadCycle : TON;
	randomUpdate : DRAND;
	valueGenerateRand : LREAL;
	percentVariation : LREAL := 0.05;
	
	
	Real_PowerA : LREAL := 1000;
	Real_PowerB : LREAL := 1000;
	Real_PowerC : LREAL := 1000;
	Real_PowerTotal : LREAL := 1000;
	Reactive_PowerA : LREAL := 1000;
	Reactive_PowerB : LREAL := 1000; 
	Reactive_PowerC : LREAL := 1000;
	Reactive_PowerTotal : LREAL := 1000;
	Apparent_PowerA : LREAL := 1000;
	Apparent_PowerB : LREAL := 1000;
	Apparent_PowerC : LREAL := 1000;
	Apparent_PowerTotal : LREAL := 1000;
	Voltage_AB : LREAL := 380;
	Voltage_BC : LREAL := 390;
	Voltage_CA : LREAL := 375;
	Voltage_LLAvg : LREAL := 382;
	Voltage_AN : LREAL := 225;
	Voltage_BN : LREAL := 230;
	Voltage_CN : LREAL := 220;
	Voltage_LNAvg : LREAL := 222;
	THDF_Voltage_AB : LREAL := 50;
	THDF_Voltage_BC : LREAL := 50;
	THDF_Voltage_CA : LREAL := 50;
	THDF_Voltage_LL : LREAL := 50;
	THDF_Voltage_AN : LREAL := 50;
	THDF_Voltage_BN : LREAL := 50;
	THDF_Voltage_CN : LREAL := 50;
	THDF_Voltage_LN : LREAL := 50;
	thdR_Voltage_AB : LREAL := 50;
	thdR_Voltage_BC : LREAL := 50;
	thdR_Voltage_CA : LREAL := 50;
	thdR_Voltage_LL : LREAL := 50;
	thdR_Voltage_AN : LREAL := 50;
	thdR_Voltage_BN : LREAL := 50;
	thdR_Voltage_CN : LREAL := 50;
	thdR_Voltage_LN : LREAL := 50;
	Current_A : LREAL := 1;
	Current_B : LREAL := 1;
	Current_C : LREAL := 1;
	Current_N : LREAL := 1;
	Current_G : LREAL := 1;
	Current_Avg : LREAL := 1;
	THDF_Current_A : LREAL := 1;
	THDF_Current_B : LREAL := 1;
	THDF_Current_C : LREAL := 1;
	THDF_Current_N : LREAL := 1 ;
	THDF_Current_G : LREAL := 1;
	thdR_Current_A : LREAL := 1;
	thdR_Current_B : LREAL := 1;
	thdR_Current_C : LREAL := 1;
	thdR_Current_N : LREAL := 1;
	thdR_Current_G : LREAL := 1;
	Total_Demand_Distortion : LREAL := 1;
	RealEnergy_IntoLoad : LREAL := 1;
	dentalRealEnergy_IntoLoad : LREAL := 1;
	RealEnergy_OutLoad : LREAL := 1;
	RealEnergy_Absolute : LREAL := 1;
	RealEnergy_Signed : LREAL := 1;
	ReactiveEnergy_IntoLoad : LREAL := 1;
	ReactiveEnergy_OutLoad : LREAL := 1;
	ReactiveEnergy_Absolute : LREAL := 1;
	ReactiveEnergy_Signed : LREAL := 1;
	ApparentEnergy_IntoLoad : LREAL := 1;
	ApparentEnergy_OutLoad : LREAL := 1;
	ApparentEnergy : LREAL := 1;
	ApparentEnergy_Delivered_Received : LREAL := 1;
	Frequency : LREAL := 50;
	PowerFactor : LREAL := 1;
	SeedDrand : INT;
	valid : BOOL;
	ProbabilityOfErrorData : LREAL := 0.1; //10%
END_VAR
VAR_STAT
	NumInstant : INT;
END_VAR
VAR PERSISTENT
	validEnvergyIntoLoad : LREAL;
END_VAR
(*VAR_IN_OUT
	PM		:	ST_PowerMeter;
END_VAR*)
VAR
	bOtherDataGood : BOOL;
END_VAR

IF bFirstCycle THEN
	bFirstCycle := FALSE;
	Param REF=  PM.Basic;
	Param.RealEnergy_IntoLoad := RealEnergy_IntoLoad;
	Param.RealEnergy_OutLoad := RealEnergy_OutLoad;
	Param.ReactiveEnergy_IntoLoad := ReactiveEnergy_IntoLoad;
	Param.ReactiveEnergy_OutLoad := ReactiveEnergy_OutLoad;
END_IF
tonReadCycle(IN := TRUE,
				PT := T#5M);

randomUpdate();
CASE estate OF
	PM_SIMU_WAIT:
		IF tonReadCycle.Q THEN
			tonReadCycle(IN:= FALSE);
			randomUpdate(Num => valueGenerateRand,
							Seed := SeedDrand);
			IF randomUpdate.Num > ProbabilityOfErrorData THEN
				estate := PM_SIMU_UPDATE;
			ELSE
				estate := PM_SIMU_READ_FAULT;
			END_IF
		END_IF
		
	PM_SIMU_UPDATE:
		Param.Real_PowerA := FgenerateRandom(percent := percentVariation, rawValue := Real_PowerA, ValueDrandGenerate := valueGenerateRand);
		Param.Real_PowerB :=  FgenerateRandom(percent := percentVariation, rawValue := Real_PowerB, ValueDrandGenerate := valueGenerateRand);
		Param.Real_PowerC := FgenerateRandom(percent := percentVariation, rawValue := Real_PowerC, ValueDrandGenerate := valueGenerateRand);
		Param.Real_PowerTotal := FgenerateRandom(percent := percentVariation, rawValue := Real_PowerTotal, ValueDrandGenerate := valueGenerateRand);
		Param.Voltage_AB := FgenerateRandom(percent := percentVariation, rawValue := Voltage_AB, ValueDrandGenerate := valueGenerateRand);
		Param.Voltage_BC := FgenerateRandom(percent := percentVariation, rawValue := Voltage_BC, ValueDrandGenerate := valueGenerateRand);
		Param.Voltage_CA := FgenerateRandom(percent := percentVariation, rawValue := Voltage_CA, ValueDrandGenerate := valueGenerateRand);
		Param.Voltage_LLAvg := FgenerateRandom(percent := percentVariation, rawValue := Voltage_LLAvg, ValueDrandGenerate := valueGenerateRand);
		Param.Voltage_AN := FgenerateRandom(percent := percentVariation, rawValue := Voltage_AN, ValueDrandGenerate := valueGenerateRand);
		Param.Voltage_BN := FgenerateRandom(percent := percentVariation, rawValue := Voltage_BN, ValueDrandGenerate := valueGenerateRand);
		Param.Voltage_CN := FgenerateRandom(percent := percentVariation, rawValue := Voltage_CN, ValueDrandGenerate := valueGenerateRand);
		Param.Voltage_LNAvg := FgenerateRandom(percent := percentVariation, rawValue := Real_PowerA, ValueDrandGenerate := valueGenerateRand);
		Param.THDF_Voltage_AB := FgenerateRandom(percent := percentVariation, rawValue := Voltage_LNAvg, ValueDrandGenerate := valueGenerateRand);
		Param.THDF_Voltage_BC := FgenerateRandom(percent := percentVariation, rawValue := THDF_Voltage_BC, ValueDrandGenerate := valueGenerateRand);
		Param.THDF_Voltage_CA := FgenerateRandom(percent := percentVariation, rawValue := THDF_Voltage_CA, ValueDrandGenerate := valueGenerateRand);
		Param.THDF_Voltage_LN := FgenerateRandom(percent := percentVariation, rawValue := THDF_Voltage_LN, ValueDrandGenerate := valueGenerateRand);
		Param.Current_A := FgenerateRandom(percent := percentVariation, rawValue := Current_A, ValueDrandGenerate := valueGenerateRand);
		Param.Current_B := FgenerateRandom(percent := percentVariation, rawValue := Current_B, ValueDrandGenerate := valueGenerateRand);
		Param.Current_C := FgenerateRandom(percent := percentVariation, rawValue := Real_PowerA, ValueDrandGenerate := valueGenerateRand);
		Param.Current_Avg := FgenerateRandom(percent := percentVariation, rawValue := Current_C, ValueDrandGenerate := valueGenerateRand);
		Param.THDF_Current_A := FgenerateRandom(percent := percentVariation, rawValue := THDF_Current_A, ValueDrandGenerate := valueGenerateRand);
		Param.THDF_Current_B := FgenerateRandom(percent := percentVariation, rawValue := THDF_Current_B, ValueDrandGenerate := valueGenerateRand);
		Param.THDF_Current_C := FgenerateRandom(percent := percentVariation, rawValue := THDF_Current_C, ValueDrandGenerate := valueGenerateRand);
		Param.THDF_Current_N := FgenerateRandom(percent := percentVariation, rawValue := THDF_Current_N, ValueDrandGenerate := valueGenerateRand);
		//
		RealEnergy_IntoLoad := RealEnergy_IntoLoad + FgenerateRandom(percent := percentVariation, rawValue := dentalRealEnergy_IntoLoad, ValueDrandGenerate := valueGenerateRand);
		Param.RealEnergy_IntoLoad := RealEnergy_IntoLoad;
		//
		Param.RealEnergy_OutLoad := RealEnergy_OutLoad + FgenerateRandom(percent := percentVariation, rawValue := 10, ValueDrandGenerate := valueGenerateRand);
		Param.ReactiveEnergy_IntoLoad := ReactiveEnergy_IntoLoad + Param.ReactiveEnergy_IntoLoad + FgenerateRandom(percent := 10, rawValue := ReactiveEnergy_IntoLoad, ValueDrandGenerate := valueGenerateRand);
		Param.ReactiveEnergy_OutLoad := ReactiveEnergy_OutLoad + FgenerateRandom(percent := percentVariation, rawValue := 10, ValueDrandGenerate := valueGenerateRand);
		Param.ApparentEnergy_IntoLoad := ApparentEnergy_IntoLoad + FgenerateRandom(percent := percentVariation, rawValue := 10, ValueDrandGenerate := valueGenerateRand);
		Param.ApparentEnergy_OutLoad := ApparentEnergy_OutLoad  + FgenerateRandom(percent := percentVariation, rawValue := 10, ValueDrandGenerate := valueGenerateRand);
		Param.PowerFactor := FgenerateRandom(percent := percentVariation, rawValue := PowerFactor, ValueDrandGenerate := valueGenerateRand);
		Param.Frequency :=  FgenerateRandom(percent := percentVariation, rawValue := Frequency, ValueDrandGenerate := valueGenerateRand);
		estate := PM_SIMU_WAIT;
				bOtherdataGood := 	IsGoodData( param.Voltage_LLAvg )
				AND IsGoodData( param.Current_Avg)
				AND IsGoodData(	param.Frequency)
				AND IsGoodData( param.Voltage_AN)
				AND IsGoodData(	param.Voltage_AB)
				AND IsGoodData( param.Voltage_BN)
				AND IsGoodData(	param.Voltage_BC)
				AND IsGoodData( param.Voltage_CN)
				AND IsGoodData(	param.Voltage_CA);
				
				
		IF IsGoodData (param.RealEnergy_IntoLoad ) AND bOtherDataGood THEN
			;// pm.Basic.RealEnergy_IntoLoad still it
			validEnvergyIntoLoad := param.RealEnergy_IntoLoad;
		ELSE
			param.RealEnergy_IntoLoad := validEnvergyIntoLoad;
		END_IF
		
		//round value
			(*param.RealEnergy_IntoLoad := F_RoundLrealEx(	lrIn 	:= param.RealEnergy_IntoLoad,
												iPrecision 	:= 0);*)
														
			param.PowerFactor := F_RoundLrealEx(	lrIn 	:= param.PowerFactor,
										iPrecision 	:= 2);
	PM_SIMU_READ_FAULT:
		param.Current_Unbalane_A := bmsConst.vINIT;
		param.Current_Unbalane_B := bmsConst.vINIT;
		param.Current_Unbalane_C := bmsConst.vINIT;
		param.Current_Unbalane_Worst := bmsConst.vINIT;
		param.Current_Unbalane_AB := bmsConst.vINIT;
		param.Current_Unbalane_BC := bmsConst.vINIT;
		param.Current_Unbalane_CA := bmsConst.vINIT;
		param.Current_Unbalane_LL_Worst := bmsConst.vINIT;
		param.Current_Unbalane_AN := bmsConst.vINIT;
		param.Current_Unbalane_BN := bmsConst.vINIT;
		param.Current_Unbalane_CN := bmsConst.vINIT;
		param.Current_Unbalane_LN_Worst := bmsConst.vINIT;
		param.Real_PowerA := bmsConst.vINIT;
		param.Real_PowerB := bmsConst.vINIT;
		param.Real_PowerC := bmsConst.vINIT;
		param.Real_PowerTotal := bmsConst.vINIT;
		param.Reactive_PowerA := bmsConst.vINIT;
		param.Reactive_PowerB := bmsConst.vINIT;
		param.Reactive_PowerC := bmsConst.vINIT;
		param.Reactive_PowerTotal := bmsConst.vINIT;
		param.Apparent_PowerA := bmsConst.vINIT;
		param.Apparent_PowerB := bmsConst.vINIT;
		param.Apparent_PowerC := bmsConst.vINIT;
		param.Apparent_PowerTotal := bmsConst.vINIT;
		param.Voltage_AB := bmsConst.vINIT;
		param.Voltage_BC := bmsConst.vINIT;
		param.Voltage_CA := bmsConst.vINIT;
		param.Voltage_LLAvg := bmsConst.vINIT;
		param.Voltage_AN := bmsConst.vINIT;
		param.Voltage_BN := bmsConst.vINIT;
		param.Voltage_CN := bmsConst.vINIT;
		param.Voltage_LNAvg := bmsConst.vINIT;
		param.THDF_Voltage_AB := bmsConst.vINIT;
		param.THDF_Voltage_BC := bmsConst.vINIT;
		param.THDF_Voltage_CA := bmsConst.vINIT;
		param.THDF_Voltage_LL := bmsConst.vINIT;
		param.THDF_Voltage_AN := bmsConst.vINIT;
		param.THDF_Voltage_BN := bmsConst.vINIT;
		param.THDF_Voltage_CN := bmsConst.vINIT;
		param.THDF_Voltage_LN := bmsConst.vINIT;
		param.thdR_Voltage_AB := bmsConst.vINIT;
		param.thdR_Voltage_BC := bmsConst.vINIT;
		param.thdR_Voltage_CA := bmsConst.vINIT;
		param.thdR_Voltage_LL := bmsConst.vINIT;
		param.thdR_Voltage_AN := bmsConst.vINIT;
		param.thdR_Voltage_BN := bmsConst.vINIT;
		param.thdR_Voltage_CN := bmsConst.vINIT;
		param.thdR_Voltage_LN := bmsConst.vINIT;
		param.Current_A := bmsConst.vINIT;
		param.Current_B := bmsConst.vINIT;
		param.Current_C := bmsConst.vINIT;
		param.Current_N := bmsConst.vINIT;
		param.Current_G := bmsConst.vINIT;
		param.Current_Avg := bmsConst.vINIT;
		param.THDF_Current_A := bmsConst.vINIT;
		param.THDF_Current_B := bmsConst.vINIT;
		param.THDF_Current_C := bmsConst.vINIT;
		param.THDF_Current_N := bmsConst.vINIT;
		param.THDF_Current_G := bmsConst.vINIT;
		param.thdR_Current_A := bmsConst.vINIT;
		param.thdR_Current_B := bmsConst.vINIT;
		param.thdR_Current_C := bmsConst.vINIT;
		param.thdR_Current_N := bmsConst.vINIT;
		param.thdR_Current_G := bmsConst.vINIT;
		param.Total_Demand_Distortion := bmsConst.vINIT;
		param.RealEnergy_IntoLoad := bmsConst.vINIT;
		param.RealEnergy_OutLoad := bmsConst.vINIT;
		param.RealEnergy_Absolute := bmsConst.vINIT;
		param.RealEnergy_Signed := bmsConst.vINIT;
		param.ReactiveEnergy_IntoLoad := bmsConst.vINIT;
		param.ReactiveEnergy_OutLoad := bmsConst.vINIT;
		param.ReactiveEnergy_Absolute := bmsConst.vINIT;
		param.ReactiveEnergy_Signed := bmsConst.vINIT;
		param.ApparentEnergy_IntoLoad := bmsConst.vINIT;
		param.ApparentEnergy_OutLoad := bmsConst.vINIT;
		param.ApparentEnergy := bmsConst.vINIT;
		param.ApparentEnergy_Delivered_Received := bmsConst.vINIT;
		param.Frequency := bmsConst.vINIT;
		param.PowerFactor := bmsConst.vINIT;

		estate := PM_SIMU_WAIT;
		
		bOtherdataGood := 	IsGoodData( param.Voltage_LLAvg )
				AND IsGoodData( param.Current_Avg)
				AND IsGoodData(	param.Frequency)
				AND IsGoodData( param.Voltage_AN)
				AND IsGoodData(	param.Voltage_AB)
				AND IsGoodData( param.Voltage_BN)
				AND IsGoodData(	param.Voltage_BC)
				AND IsGoodData( param.Voltage_CN)
				AND IsGoodData(	param.Voltage_CA);
				
				
	IF IsGoodData (param.RealEnergy_IntoLoad ) AND bOtherDataGood THEN
		;// pm.Basic.RealEnergy_IntoLoad still it
		validEnvergyIntoLoad := param.RealEnergy_IntoLoad;
	ELSE
		param.RealEnergy_IntoLoad := validEnvergyIntoLoad;
	END_IF
	
	//round value
		(*param.RealEnergy_IntoLoad := F_RoundLrealEx(	lrIn 	:= param.RealEnergy_IntoLoad,
											iPrecision 	:= 0);*)
													
		param.PowerFactor := F_RoundLrealEx(	lrIn 	:= param.PowerFactor,
									iPrecision 	:= 2);
	
END_CASE

METHOD Constructor : BOOL
VAR_INPUT
END_VAR
NumInstant := NumInstant + 1;
SeedDrand := NumInstant;
END_METHOD

PROPERTY Name : string
GET
Name := sName;
END_GET
SET
sName := Name;
END_SET
END_PROPERTY

PROPERTY p_ApparentEnergy_IntoLoad : Lreal
GET
p_ApparentEnergy_IntoLoad := ApparentEnergy_IntoLoad;
END_GET
SET
ApparentEnergy_IntoLoad := p_ApparentEnergy_IntoLoad  ;
END_SET
END_PROPERTY

PROPERTY p_ApparentEnergy_OutLoad : Lreal
GET
END_GET
SET
ApparentEnergy_OutLoad := p_ApparentEnergy_OutLoad;
END_SET
END_PROPERTY

PROPERTY p_Current_A : Lreal
GET
END_GET
SET
Current_A := p_Current_A;
END_SET
END_PROPERTY

PROPERTY p_Current_Avg : Lreal
GET
END_GET
SET
Current_Avg := p_Current_Avg;
END_SET
END_PROPERTY

PROPERTY p_Current_B : Lreal
GET
END_GET
SET
Current_B := p_Current_B;
END_SET
END_PROPERTY

PROPERTY p_Current_C : Lreal
GET
END_GET
SET
Current_C := p_Current_C;
END_SET
END_PROPERTY

PROPERTY p_dentalRealEnergy_IntoLoad : Lreal
GET
END_GET
SET
dentalRealEnergy_IntoLoad := p_dentalRealEnergy_IntoLoad;
END_SET
END_PROPERTY

PROPERTY p_PowerFactor : Lreal
GET
END_GET
SET
PowerFactor := p_PowerFactor;
END_SET
END_PROPERTY

PROPERTY p_ReactiveEnergy_IntoLoad : Lreal
GET
END_GET
SET
ReactiveEnergy_IntoLoad := p_ReactiveEnergy_IntoLoad;
END_SET
END_PROPERTY

PROPERTY p_ReactiveEnergy_OutLoad : Lreal
GET
END_GET
SET
ReactiveEnergy_OutLoad := p_ReactiveEnergy_OutLoad;
END_SET
END_PROPERTY

PROPERTY p_Real_PowerA : Lreal
GET
END_GET
SET
Real_PowerA := p_Real_PowerA;
END_SET
END_PROPERTY

PROPERTY p_Real_PowerB : Lreal
GET
END_GET
SET
Real_PowerB := p_Real_PowerB;
END_SET
END_PROPERTY

PROPERTY p_Real_PowerC : Lreal
GET
END_GET
SET
Real_PowerC := p_Real_PowerC;
END_SET
END_PROPERTY

PROPERTY p_Real_PowerTotal : Lreal
GET
END_GET
SET
Real_PowerTotal := p_Real_PowerTotal;
END_SET
END_PROPERTY

PROPERTY p_RealEnergy_IntoLoad : Lreal
GET
p_RealEnergy_IntoLoad := RealEnergy_IntoLoad;
END_GET
SET
RealEnergy_IntoLoad := p_RealEnergy_IntoLoad;
END_SET
END_PROPERTY

PROPERTY p_RealEnergy_OutLoad : Lreal
GET
END_GET
SET
RealEnergy_OutLoad := p_RealEnergy_OutLoad;
END_SET
END_PROPERTY

PROPERTY Ref_PM : Reference to ST_PowerMeter
GET
END_GET
SET
PM Ref= Ref_PM;
END_SET
END_PROPERTY

END_FUNCTION_BLOCK

// ---- TEST/PgrTest.TcPOU
PROGRAM PgrTest
VAR
	arPM : ARRAY[0..NumRealMeters-1] OF FB_PmSimulate;
	bFirstCycle : BOOL := true;
	iloop : UINT;

END_VAR
VAR CONSTANT
	NumRealMeters : UINT := 72;
	arDentalRealEnergy_IntoLoad : ARRAY[0..NumRealMeters-1] OF LREAL := [	81.4864739239071,
																				80.361624988331,
																				0,
																				3.43962071209237,
																				7.61364692757743,
																				7.02333364320482,
																				0,
																				1.16203402435553,
																				1.98010597750182,
																				3.70456446964543,
																				0,
																				0,
																				0,
																				0.599609556567453,
																				0,
																				0,
																				0,
																				96.1931765361507,
																				39.2256205261452,
																				48.2615970995338,
																				8.1342381704887,
																				0,
																				0,
																				0,
																				0,
																				0,
																				0,
																				14.678813795659,
																				0,
																				5.05717207399526,
																				14.8229060146791,
																				11.550618202094,
																				0,
																				0,
																				0,
																				0,
																				0,
																				1.58036627312352,
																				0,
																				0.460165473644789,
																				0.469461745839634,
																				0.0511294970716433,
																				0.57172073998292,
																				60.4118248581952,
																				30.0594961420288,
																				18.4763409872529,
																				2.66338198382287,
																				0.515943106813855,
																				0.260295621455638,
																				2.56577112577701,
																				1.849958166774,
																				2.35195686529559,
																				1.20386724923233,
																				1.7662917170204,
																				1.56177372873383,
																				5.14083852374886,
																				31.3144928883328,
																				31.0449009946823,
																				2.16138328530128,
																				2.62154875894607,
																				4.88054290229322,
																				8.05521985683253,
																				0.492702426326744,
																				0.952867899971534,
																				2.31012364041879,
																				7.18601840661459,
																				11.6575253323347,
																				1.99869852189151,
																				0.134795946825241,
																				0.488054290229322,
																				0.0278888165845327,
																				0.0139444082922663
																				];


END_VAR
VAR PERSISTENT 
	
	LV01_Real_RealEnergy_IntoLoad : LREAL := 3630639; 
	DB_PR1_1_Real_RealEnergy_IntoLoad : LREAL := 14149755;
	DB1_Real_RealEnergy_IntoLoad : LREAL := 6246714;
	DB2_Real_RealEnergy_IntoLoad : LREAL := 4873554;
	DB3_Real_RealEnergy_IntoLoad : LREAL := 6891408;
	DB4_Real_RealEnergy_IntoLoad : LREAL := 6437618;
	DB1_1_Real_RealEnergy_IntoLoad : LREAL :=  0;
	DB2_1_Real_RealEnergy_IntoLoad : LREAL := 1551326;
	DB3_1_Real_RealEnergy_IntoLoad : LREAL := 1557420;
	DB4_1_Real_RealEnergy_IntoLoad : LREAL :=  722266;
	DB5_Real_RealEnergy_IntoLoad : LREAL :=  16192073;
	DB6_Real_RealEnergy_IntoLoad : LREAL := 16830162;
	DB7_Real_RealEnergy_IntoLoad : LREAL :=  16947698;
	DB_MR_Real_RealEnergy_IntoLoad : LREAL :=  1225028;
	DB5_1_Real_RealEnergy_IntoLoad : LREAL := 0;
	DB6_1_Real_RealEnergy_IntoLoad : LREAL :=  0;
	DB7_1_Real_RealEnergy_IntoLoad : LREAL := 0;
	LV02_Real_RealEnergy_IntoLoad : LREAL := 6829629;
	DB_PR1_2_Real_RealEnergy_IntoLoad : LREAL := 8091123;
	DB_AIRCOMP_Real_RealEnergy_IntoLoad : LREAL := 7697622;
	DB_AHU_Real_RealEnergy_IntoLoad : LREAL := 12769798;
	DB8_Real_RealEnergy_IntoLoad : LREAL := 17048080;
	DB9_Real_RealEnergy_IntoLoad : LREAL := 16994216;
	DB10_Real_RealEnergy_IntoLoad : LREAL :=  6143691;
	DB8_1_Real_RealEnergy_IntoLoad : LREAL :=  0;
	DB9_1_Real_RealEnergy_IntoLoad : LREAL := 0;
	DB10_1_Real_RealEnergy_IntoLoad : LREAL := 0;
	A1_Real_RealEnergy_IntoLoad : LREAL := 491971;
	A2_Real_RealEnergy_IntoLoad : LREAL :=  659353;
	A3_Real_RealEnergy_IntoLoad : LREAL := 367659;
	A4_Real_RealEnergy_IntoLoad : LREAL := 410530;
	A5_Real_RealEnergy_IntoLoad : LREAL :=  708399;
	LP_PR1A_Real_RealEnergy_IntoLoad : LREAL := 0;
	LP_PR1B_Real_RealEnergy_IntoLoad : LREAL := 0;
	LP_PR2A_Real_RealEnergy_IntoLoad : LREAL := 0;
	LP_PR2B_Real_RealEnergy_IntoLoad : LREAL := 0;
	LP_PR3A_Real_RealEnergy_IntoLoad : LREAL := 0;
	DB_WH_Real_RealEnergy_IntoLoad : LREAL := 3215883;
	LP_PR3B_Real_RealEnergy_IntoLoad : LREAL := 0;
	LP_PR4A_Real_RealEnergy_IntoLoad : LREAL :=  344117;
	LP_PR4B_Real_RealEnergy_IntoLoad : LREAL := 356961;
	LP_BM_Real_RealEnergy_IntoLoad : LREAL := 129467;
	DB_BM_Real_RealEnergy_IntoLoad : LREAL := 837274;
	LV03_Real_RealEnergy_IntoLoad : LREAL := 9800613;
	DB_MVAC1_Real_RealEnergy_IntoLoad : LREAL := 6100039;
	DB_MVAC2_Real_RealEnergy_IntoLoad : LREAL := 2814844;
	DB_OFF2_Real_RealEnergy_IntoLoad : LREAL :=  4121718;
	LP_EL1_Real_RealEnergy_IntoLoad : LREAL :=  89440;
	LP_EL2_Real_RealEnergy_IntoLoad : LREAL :=  676522;
	DB_OFF1_Real_RealEnergy_IntoLoad : LREAL := 3137595;
	DB_KIT_Real_RealEnergy_IntoLoad : LREAL := 2163140;
	LP_WH2_Real_RealEnergy_IntoLoad : LREAL := 1905378;
	LP_WH1_Real_RealEnergy_IntoLoad : LREAL := 192677;
	CH4_Real_RealEnergy_IntoLoad : LREAL := 180401;
	CH5_Real_RealEnergy_IntoLoad : LREAL := 126235;
	CH6_Real_RealEnergy_IntoLoad : LREAL := 225603;
	LV04_Real_RealEnergy_IntoLoad : LREAL := 4422056;
	DB_PR2_Real_RealEnergy_IntoLoad : LREAL := 31131722;
	DB11_Real_RealEnergy_IntoLoad : LREAL := 2658776;
	DB12_Real_RealEnergy_IntoLoad : LREAL := 3431708;
	DB13_Real_RealEnergy_IntoLoad : LREAL :=  4640308;
	DB14_Real_RealEnergy_IntoLoad : LREAL := 7195837;
	DB11_1_Real_RealEnergy_IntoLoad : LREAL := 575609;
	DB12_1_Real_RealEnergy_IntoLoad : LREAL := 1252745;
	DB13_1_Real_RealEnergy_IntoLoad : LREAL := 1380059;
	DB14_1_Real_RealEnergy_IntoLoad : LREAL := 3846554;
	DB15_Real_RealEnergy_IntoLoad : LREAL := 7943089;
	DB15_1_Real_RealEnergy_IntoLoad : LREAL := 4303139;
	LP_PR5A_Real_RealEnergy_IntoLoad : LREAL := 124750;
	LP_PR5B_Real_RealEnergy_IntoLoad : LREAL := 275030;
	LP_PR6A_Real_RealEnergy_IntoLoad : LREAL := 30196;
	LP_PR6B_Real_RealEnergy_IntoLoad : LREAL := 22547;

END_VAR

IF bFirstCycle THEN
	bFirstCycle := FALSE;
	FirstCycle();
END_IF

FOR iloop := 0 TO NumRealMeters-1 DO 
	// fb processing
	arPM[iloop]();
	// return Real_RealEnergy_IntoLoad
	LV01_Real_RealEnergy_IntoLoad := arPM[LV01].p_RealEnergy_IntoLoad;
	DB_PR1_1_Real_RealEnergy_IntoLoad := arPM[DB_PR1_1].p_RealEnergy_IntoLoad;
	DB1_Real_RealEnergy_IntoLoad := arPM[DB1].p_RealEnergy_IntoLoad;
	DB2_Real_RealEnergy_IntoLoad := arPM[DB2].p_RealEnergy_IntoLoad;
	DB3_Real_RealEnergy_IntoLoad := arPM[DB3].p_RealEnergy_IntoLoad;
	DB4_Real_RealEnergy_IntoLoad := arPM[DB4].p_RealEnergy_IntoLoad;
	DB1_1_Real_RealEnergy_IntoLoad := arPM[DB1_1].p_RealEnergy_IntoLoad;
	DB2_1_Real_RealEnergy_IntoLoad := arPM[DB2_1].p_RealEnergy_IntoLoad;
	DB3_1_Real_RealEnergy_IntoLoad := arPM[DB3_1].p_RealEnergy_IntoLoad;
	DB4_1_Real_RealEnergy_IntoLoad := arPM[DB4_1].p_RealEnergy_IntoLoad;
	DB5_Real_RealEnergy_IntoLoad := arPM[DB5].p_RealEnergy_IntoLoad;
	DB6_Real_RealEnergy_IntoLoad := arPM[DB6].p_RealEnergy_IntoLoad;
	DB7_Real_RealEnergy_IntoLoad := arPM[DB7].p_RealEnergy_IntoLoad;
	DB_MR_Real_RealEnergy_IntoLoad := arPM[DB_MR].p_RealEnergy_IntoLoad;
	DB5_1_Real_RealEnergy_IntoLoad := arPM[DB5_1].p_RealEnergy_IntoLoad;
	DB6_1_Real_RealEnergy_IntoLoad := arPM[DB6_1].p_RealEnergy_IntoLoad;
	DB7_1_Real_RealEnergy_IntoLoad := arPM[DB7_1].p_RealEnergy_IntoLoad;
	LV02_Real_RealEnergy_IntoLoad := arPM[LV02].p_RealEnergy_IntoLoad;
	DB_PR1_2_Real_RealEnergy_IntoLoad := arPM[DB_PR1_2].p_RealEnergy_IntoLoad;
	DB_AIRCOMP_Real_RealEnergy_IntoLoad := arPM[DB_AIRCOMP].p_RealEnergy_IntoLoad;
	DB_AHU_Real_RealEnergy_IntoLoad := arPM[DB_AHU].p_RealEnergy_IntoLoad;
	DB8_Real_RealEnergy_IntoLoad := arPM[DB8].p_RealEnergy_IntoLoad;
	DB9_Real_RealEnergy_IntoLoad := arPM[DB9].p_RealEnergy_IntoLoad;
	DB10_Real_RealEnergy_IntoLoad := arPM[DB10].p_RealEnergy_IntoLoad;
	DB8_1_Real_RealEnergy_IntoLoad := arPM[DB8_1].p_RealEnergy_IntoLoad;
	DB9_1_Real_RealEnergy_IntoLoad := arPM[DB9_1].p_RealEnergy_IntoLoad;
	DB10_1_Real_RealEnergy_IntoLoad := arPM[DB10_1].p_RealEnergy_IntoLoad;
	A1_Real_RealEnergy_IntoLoad := arPM[A1].p_RealEnergy_IntoLoad;
	A2_Real_RealEnergy_IntoLoad := arPM[A2].p_RealEnergy_IntoLoad;
	A3_Real_RealEnergy_IntoLoad := arPM[A3].p_RealEnergy_IntoLoad;
	A4_Real_RealEnergy_IntoLoad := arPM[A4].p_RealEnergy_IntoLoad;
	A5_Real_RealEnergy_IntoLoad := arPM[A5].p_RealEnergy_IntoLoad;
	LP_PR1A_Real_RealEnergy_IntoLoad := arPM[LP_PR1A].p_RealEnergy_IntoLoad;
	LP_PR1B_Real_RealEnergy_IntoLoad := arPM[LP_PR1B].p_RealEnergy_IntoLoad;
	LP_PR2A_Real_RealEnergy_IntoLoad := arPM[LP_PR2A].p_RealEnergy_IntoLoad;
	LP_PR2B_Real_RealEnergy_IntoLoad := arPM[LP_PR2B].p_RealEnergy_IntoLoad;
	LP_PR3A_Real_RealEnergy_IntoLoad := arPM[LP_PR3A].p_RealEnergy_IntoLoad;
	DB_WH_Real_RealEnergy_IntoLoad := arPM[DB_WH].p_RealEnergy_IntoLoad;
	LP_PR3B_Real_RealEnergy_IntoLoad := arPM[LP_PR3B].p_RealEnergy_IntoLoad;
	LP_PR4A_Real_RealEnergy_IntoLoad := arPM[LP_PR4A].p_RealEnergy_IntoLoad;
	LP_PR4B_Real_RealEnergy_IntoLoad := arPM[LP_PR4B].p_RealEnergy_IntoLoad;
	LP_BM_Real_RealEnergy_IntoLoad := arPM[LP_BM].p_RealEnergy_IntoLoad;
	DB_BM_Real_RealEnergy_IntoLoad := arPM[DB_BM].p_RealEnergy_IntoLoad;
	LV03_Real_RealEnergy_IntoLoad := arPM[LV03].p_RealEnergy_IntoLoad;
	DB_MVAC1_Real_RealEnergy_IntoLoad := arPM[DB_MVAC1].p_RealEnergy_IntoLoad;
	DB_MVAC2_Real_RealEnergy_IntoLoad := arPM[DB_MVAC2].p_RealEnergy_IntoLoad;
	DB_OFF2_Real_RealEnergy_IntoLoad := arPM[DB_OFF2].p_RealEnergy_IntoLoad;
	LP_EL1_Real_RealEnergy_IntoLoad := arPM[LP_EL1].p_RealEnergy_IntoLoad;
	LP_EL2_Real_RealEnergy_IntoLoad := arPM[LP_EL2].p_RealEnergy_IntoLoad;
	DB_OFF1_Real_RealEnergy_IntoLoad := arPM[DB_OFF1].p_RealEnergy_IntoLoad;
	DB_KIT_Real_RealEnergy_IntoLoad := arPM[DB_KIT].p_RealEnergy_IntoLoad;
	LP_WH2_Real_RealEnergy_IntoLoad := arPM[LP_WH2].p_RealEnergy_IntoLoad;
	LP_WH1_Real_RealEnergy_IntoLoad := arPM[LP_WH1].p_RealEnergy_IntoLoad;
	CH4_Real_RealEnergy_IntoLoad := arPM[CH4].p_RealEnergy_IntoLoad;
	CH5_Real_RealEnergy_IntoLoad := arPM[CH5].p_RealEnergy_IntoLoad;
	CH6_Real_RealEnergy_IntoLoad := arPM[CH6].p_RealEnergy_IntoLoad;
	LV04_Real_RealEnergy_IntoLoad := arPM[LV04].p_RealEnergy_IntoLoad;
	DB_PR2_Real_RealEnergy_IntoLoad := arPM[DB_PR2].p_RealEnergy_IntoLoad;
	DB11_Real_RealEnergy_IntoLoad := arPM[DB11].p_RealEnergy_IntoLoad;
	DB12_Real_RealEnergy_IntoLoad := arPM[DB12].p_RealEnergy_IntoLoad;
	DB13_Real_RealEnergy_IntoLoad := arPM[DB13].p_RealEnergy_IntoLoad;
	DB14_Real_RealEnergy_IntoLoad := arPM[DB14].p_RealEnergy_IntoLoad;
	DB11_1_Real_RealEnergy_IntoLoad := arPM[DB11_1].p_RealEnergy_IntoLoad;
	DB12_1_Real_RealEnergy_IntoLoad := arPM[DB12_1].p_RealEnergy_IntoLoad;
	DB13_1_Real_RealEnergy_IntoLoad := arPM[DB13_1].p_RealEnergy_IntoLoad;
	DB14_1_Real_RealEnergy_IntoLoad := arPM[DB14_1].p_RealEnergy_IntoLoad;
	DB15_Real_RealEnergy_IntoLoad := arPM[DB15].p_RealEnergy_IntoLoad;
	DB15_1_Real_RealEnergy_IntoLoad := arPM[DB15_1].p_RealEnergy_IntoLoad;
	LP_PR5A_Real_RealEnergy_IntoLoad := arPM[LP_PR5A].p_RealEnergy_IntoLoad;
	LP_PR5B_Real_RealEnergy_IntoLoad := arPM[LP_PR5B].p_RealEnergy_IntoLoad;
	LP_PR6A_Real_RealEnergy_IntoLoad := arPM[LP_PR6A].p_RealEnergy_IntoLoad;
	LP_PR6B_Real_RealEnergy_IntoLoad := arPM[LP_PR6B].p_RealEnergy_IntoLoad;

	
	
END_FOR

METHOD FirstCycle : BOOL
VAR_INPUT
END_VAR
VAR
	iloop : UINT;
END_VAR
// PMSimulate Constructor 
	FOR iloop := 0 TO NumRealMeters -1 DO
		arPM[iloop].Constructor();
	END_FOR
//Naming
	arPM[LV01].Name := 'LV01';
	arPM[DB_PR1_1].Name := 'DB_PR1_1';
	arPM[DB1].Name := 'DB1';
	arPM[DB2].Name := 'DB2';
	arPM[DB3].Name := 'DB3';
	arPM[DB4].Name := 'DB4';
	arPM[DB1_1].Name := 'DB1_1';
	arPM[DB2_1].Name := 'DB2_1';
	arPM[DB3_1].Name := 'DB3_1';
	arPM[DB4_1].Name := 'DB4_1';
	arPM[DB5].Name := 'DB5';
	arPM[DB6].Name := 'DB6';
	arPM[DB7].Name := 'DB7';
	arPM[DB_MR].Name := 'DB_MR';
	arPM[DB5_1].Name := 'DB5_1';
	arPM[DB6_1].Name := 'DB6_1';
	arPM[DB7_1].Name := 'DB7_1';
	arPM[LV02].Name := 'LV02';
	arPM[DB_PR1_2].Name := 'DB_PR1_2';
	arPM[DB_AIRCOMP].Name := 'DB_AIRCOMP';
	arPM[DB_AHU].Name := 'DB_AHU';
	arPM[DB8].Name := 'DB8';
	arPM[DB9].Name := 'DB9';
	arPM[DB10].Name := 'DB10';
	arPM[DB8_1].Name := 'DB8_1';
	arPM[DB9_1].Name := 'DB9_1';
	arPM[DB10_1].Name := 'DB10_1';
	arPM[A1].Name := 'A1';
	arPM[A2].Name := 'A2';
	arPM[A3].Name := 'A3';
	arPM[A4].Name := 'A4';
	arPM[A5].Name := 'A5';
	arPM[LP_PR1A].Name := 'LP_PR1A';
	arPM[LP_PR1B].Name := 'LP_PR1B';
	arPM[LP_PR2A].Name := 'LP_PR2A';
	arPM[LP_PR2B].Name := 'LP_PR2B';
	arPM[LP_PR3A].Name := 'LP_PR3A';
	arPM[DB_WH].Name := 'DB_WH';
	arPM[LP_PR3B].Name := 'LP_PR3B';
	arPM[LP_PR4A ].Name := 'LP_PR4A ';
	arPM[LP_PR4B].Name := 'LP_PR4B';
	arPM[LP_BM].Name := 'LP_BM';
	arPM[DB_BM].Name := 'DB_BM';
	arPM[LV03].Name := 'LV03';
	arPM[DB_MVAC1].Name := 'DB_MVAC1';
	arPM[DB_MVAC2].Name := 'DB_MVAC2';
	arPM[DB_OFF2].Name := 'DB_OFF2';
	arPM[LP_EL1].Name := 'LP_EL1';
	arPM[LP_EL2].Name := 'LP_EL2';
	arPM[DB_OFF1].Name := 'DB_OFF1';
	arPM[DB_KIT].Name := 'DB_KIT';
	arPM[LP_WH2].Name := 'LP_WH2';
	arPM[LP_WH1].Name := 'LP_WH1';
	arPM[CH4].Name := 'CH4';
	arPM[CH5].Name := 'CH5';
	arPM[CH6].Name := 'CH6';
	arPM[LV04].Name := 'LV04';
	arPM[DB_PR2].Name := 'DB_PR2';
	arPM[DB11].Name := 'DB11';
	arPM[DB12].Name := 'DB12';
	arPM[DB13].Name := 'DB13';
	arPM[DB14].Name := 'DB14';
	arPM[DB11_1].Name := 'DB11_1';
	arPM[DB12_1].Name := 'DB12_1';
	arPM[DB13_1].Name := 'DB13_1';
	arPM[DB14_1].Name := 'DB14_1';
	arPM[DB15].Name := 'DB15';
	arPM[DB15_1].Name := 'DB15_1';
	arPM[LP_PR5A].Name := 'LP_PR5A';
	arPM[LP_PR5B].Name := 'LP_PR5B';
	arPM[LP_PR6A].Name := 'LP_PR6A';
	arPM[LP_PR6B].Name := 'LP_PR6B';

// reference 
	arPM[LV01].Ref_PM REF= pmDev.DB07_01_5500;
	arPM[DB_PR1_1].Ref_PM REF= pmDev.DB06_06_5500;
	arPM[DB1].Ref_PM ref= pmDev.DB05_10_5500;
	arPM[DB2].Ref_PM ref= pmDev.DB04_06_5500;
	arPM[DB3].Ref_PM ref= pmDev.DB04_04_5500;
	arPM[DB4].Ref_PM ref= pmDev.DB04_02_5500;
	arPM[DB1_1].Ref_PM ref= pmDev.DB05_09_5350;
	arPM[DB2_1].Ref_PM ref= pmDev.DB04_05_5350;
	arPM[DB3_1].Ref_PM ref= pmDev.DB04_03_5350;
	arPM[DB4_1].Ref_PM ref= pmDev.DB04_01_5350;
	arPM[DB5].Ref_PM ref= pmDev.DB03_04_5500;
	arPM[DB6].Ref_PM ref= pmDev.DB03_06_5500;
	arPM[DB7].Ref_PM ref= pmDev.DB03_02_5500;
	arPM[DB_MR].Ref_PM ref= pmDev.DB06_11_5500;
	arPM[DB5_1].Ref_PM ref= pmDev.DB03_03_5350;
	arPM[DB6_1].Ref_PM ref= pmDev.DB03_05_5350;
	arPM[DB7_1].Ref_PM ref= pmDev.DB03_01_5350;
	arPM[LV02].Ref_PM ref= pmDev.DB07_02_5500;
	arPM[DB_PR1_2].Ref_PM ref= pmDev.DB06_05_5500;
	arPM[DB_AIRCOMP].Ref_PM ref= pmDev.DB07_03_5500;
	arPM[DB_AHU].Ref_PM ref= pmDev.DB06_07_5500;
	arPM[DB8].Ref_PM ref= pmDev.DB05_04_5500;
	arPM[DB9].Ref_PM ref= pmDev.DB05_06_5500;
	arPM[DB10].Ref_PM ref= pmDev.DB05_08_5500;
	arPM[DB8_1].Ref_PM ref= pmDev.DB05_03_5350;
	arPM[DB9_1].Ref_PM ref= pmDev.DB05_05_5350;
	arPM[DB10_1].Ref_PM ref= pmDev.DB05_07_5350;
	arPM[A1].Ref_PM ref= pmDev.DB07_06_5350;
	arPM[A2].Ref_PM ref= pmDev.DB07_07_5350;
	arPM[A3].Ref_PM ref= pmDev.DB07_08_5350;
	arPM[A4].Ref_PM ref= pmDev.DB07_09_5350;
	arPM[A5].Ref_PM ref= pmDev.DB07_10_5350;
	arPM[LP_PR1A].Ref_PM ref= pmDev.DB05_01_5350;
	arPM[LP_PR1B].Ref_PM ref= pmDev.DB05_02_5350;
	arPM[LP_PR2A].Ref_PM ref= pmDev.DB05_22_5350;
	arPM[LP_PR2B].Ref_PM ref= pmDev.DB05_21_5350;
	arPM[LP_PR3A].Ref_PM ref= pmDev.DB03_08_5350;
	arPM[DB_WH].Ref_PM ref= pmDev.DB01_18_5500;
	arPM[LP_PR3B].Ref_PM ref= pmDev.DB03_07_5350;
	arPM[LP_PR4A ].Ref_PM ref= pmDev.DB04_08_5350;
	arPM[LP_PR4B].Ref_PM ref= pmDev.DB04_07_5350;
	arPM[LP_BM].Ref_PM ref= pmDev.DB01_20_5500;
	arPM[DB_BM].Ref_PM ref= pmDev.DB01_22_5500;
	arPM[LV03].Ref_PM ref= pmDev.DB06_04_5500;
	arPM[DB_MVAC1].Ref_PM ref= pmDev.DB07_05_5500;
	arPM[DB_MVAC2].Ref_PM ref= pmDev.DB07_04_5500;
	arPM[DB_OFF2].Ref_PM ref= pmDev.DB06_38_5500;
	arPM[LP_EL1].Ref_PM ref= pmDev.DB06_03_5500;
	arPM[LP_EL2].Ref_PM ref= pmDev.DB06_01_5500;
	arPM[DB_OFF1].Ref_PM ref= pmDev.DB06_08_5500;
	arPM[DB_KIT].Ref_PM ref= pmDev.DB06_33_5500;
	arPM[LP_WH2].Ref_PM ref= pmDev.DB01_12_5350;
	arPM[LP_WH1].Ref_PM ref= pmDev.DB01_11_5500;
	arPM[CH4].Ref_PM ref= pmDev.DB07_11_5350;
	arPM[CH5].Ref_PM ref= pmDev.DB07_12_5350;
	arPM[CH6].Ref_PM ref= pmDev.DB07_13_5350;
	arPM[LV04].Ref_PM ref= pmDev.DB06_02_5500;
	arPM[DB_PR2].Ref_PM ref= pmDev.DB01_07_5500;
	arPM[DB11].Ref_PM ref= pmDev.DB01_04_5500;
	arPM[DB12].Ref_PM ref= pmDev.DB01_01_5500;
	arPM[DB13].Ref_PM ref= pmDev.DB02_02_5500;
	arPM[DB14].Ref_PM ref= pmDev.DB02_06_5500;
	arPM[DB11_1].Ref_PM ref= pmDev.DB01_03_5350;
	arPM[DB12_1].Ref_PM ref= pmDev.DB01_02_5350;
	arPM[DB13_1].Ref_PM ref= pmDev.DB02_01_5350;
	arPM[DB14_1].Ref_PM ref= pmDev.DB02_05_5350;
	arPM[DB15].Ref_PM ref= pmDev.DB02_04_5500;
	arPM[DB15_1].Ref_PM ref= pmDev.DB02_03_5350;
	arPM[LP_PR5A].Ref_PM ref= pmDev.DB02_08_5350;
	arPM[LP_PR5B].Ref_PM ref= pmDev.DB02_07_5350;
	arPM[LP_PR6A].Ref_PM ref= pmDev.DB01_06_5350;
	arPM[LP_PR6B].Ref_PM ref= pmDev.DB01_05_5350;
// set Current A
	arPM[LV01].p_Current_A := 1500;
	arPM[DB_PR1_1].p_Current_A := 1783 ;
	//arPM[DB1].p_Current_A := 50;
	arPM[DB2].p_Current_A :=  51;
	arPM[DB3].p_Current_A := 136;
	arPM[DB4].p_Current_A := 223;
	//arPM[DB1_1].p_Current_A := ;
	arPM[DB2_1].p_Current_A := 30;
	arPM[DB3_1].p_Current_A := 50 ;
	arPM[DB4_1].p_Current_A :=  100;
	//arPM[DB5].p_Current_A := ;
	//arPM[DB6].p_Current_A := ;
	//arPM[DB7].p_Current_A := ;
	arPM[DB_MR].p_Current_A := 10;
	//arPM[DB5_1].p_Current_A := ;
	//arPM[DB6_1].p_Current_A := ;
	//arPM[DB7_1].p_Current_A := ;
	arPM[LV02].p_Current_A := 1789;
	arPM[DB_PR1_2].p_Current_A := 884;
	arPM[DB_AIRCOMP].p_Current_A := 952;
	arPM[DB_AHU].p_Current_A := 151;
	//arPM[DB8].p_Current_A := ;
	//arPM[DB9].p_Current_A := ;
	//arPM[DB10].p_Current_A := ;
	//arPM[DB8_1].p_Current_A := ;
	//arPM[DB9_1].p_Current_A := ;
	//arPM[DB10_1].p_Current_A := ;
	arPM[A1].p_Current_A := 287 ;
	//arPM[A2].p_Current_A := ;
	arPM[A3].p_Current_A := 87 ;
	arPM[A4].p_Current_A := 297;
	arPM[A5].p_Current_A := 239;
	//arPM[LP_PR1A].p_Current_A := ;
	//arPM[LP_PR1B].p_Current_A := ;
	//arPM[LP_PR2A].p_Current_A := ;
	//arPM[LP_PR2B].p_Current_A := ;
	//arPM[LP_PR3A].p_Current_A := ;
	arPM[DB_WH].p_Current_A := 26.4;
	//arPM[LP_PR3B].p_Current_A := ;
	arPM[LP_PR4A ].p_Current_A := 8.8;
	arPM[LP_PR4B].p_Current_A := 8.5;
	arPM[LP_BM].p_Current_A := 0.4;
	arPM[DB_BM].p_Current_A := 17.68;
	arPM[LV03].p_Current_A := 1103 ;
	arPM[DB_MVAC1].p_Current_A := 596;
	arPM[DB_MVAC2].p_Current_A :=342;
	arPM[DB_OFF2].p_Current_A := 45 ;
	arPM[LP_EL1].p_Current_A := 17;
	arPM[LP_EL2].p_Current_A := 2.5;
	arPM[DB_OFF1].p_Current_A := 42.7;
	arPM[DB_KIT].p_Current_A := 20.8;
	arPM[LP_WH2].p_Current_A := 56;
	arPM[LP_WH1].p_Current_A := 19.32;
	arPM[CH4].p_Current_A := 0.86;
	arPM[CH5].p_Current_A := 77.4;
	arPM[CH6].p_Current_A := 1.6;
	arPM[LV04].p_Current_A := 602.6;
	arPM[DB_PR2].p_Current_A := 516;
	arPM[DB11].p_Current_A := 19.68;
	arPM[DB12].p_Current_A := 52.6;
	arPM[DB13].p_Current_A := 128.3;
	arPM[DB14].p_Current_A := 153.9;
	arPM[DB11_1].p_Current_A := 0.104;
	arPM[DB12_1].p_Current_A := 12.16;
	arPM[DB13_1].p_Current_A := 49.97;
	arPM[DB14_1].p_Current_A := 130.8;
	arPM[DB15].p_Current_A := 161.92;
	arPM[DB15_1].p_Current_A := 36.45;
	arPM[LP_PR5A].p_Current_A := 11.18;
	arPM[LP_PR5B].p_Current_A := 9.24;
	arPM[LP_PR6A].p_Current_A := 0.5544;
	arPM[LP_PR6B].p_Current_A := 0.29;
// CurrentB
	arPM[LV01].p_Current_B := 1458;
	arPM[DB_PR1_1].p_Current_B := 1707 ;
	//arPM[DB1].p_Current_B := 50;
	arPM[DB2].p_Current_B :=  87;
	arPM[DB3].p_Current_B := 152;
	arPM[DB4].p_Current_B := 227.4;
	//arPM[DB1_1].p_Current_B := ;
	arPM[DB2_1].p_Current_B := 32;
	arPM[DB3_1].p_Current_B := 50 ;
	arPM[DB4_1].p_Current_B :=  112;
	//arPM[DB5].p_Current_B := ;
	//arPM[DB6].p_Current_B := ;
	//arPM[DB7].p_Current_B := ;
	arPM[DB_MR].p_Current_B := 44.88;
	//arPM[DB5_1].p_Current_B := ;
	//arPM[DB6_1].p_Current_B := ;
	//arPM[DB7_1].p_Current_B := ;
	arPM[LV02].p_Current_B := 1595;
	arPM[DB_PR1_2].p_Current_B := 717;
	arPM[DB_AIRCOMP].p_Current_B := 913;
	arPM[DB_AHU].p_Current_B := 146;
	//arPM[DB8].p_Current_B := ;
	//arPM[DB9].p_Current_B := ;
	//arPM[DB10].p_Current_B := ;
	//arPM[DB8_1].p_Current_B := ;
	//arPM[DB9_1].p_Current_B := ;
	//arPM[DB10_1].p_Current_B := ;
	arPM[A1].p_Current_B := 289 ;
	//arPM[A2].p_Current_B := ;
	arPM[A3].p_Current_B := 96 ;
	arPM[A4].p_Current_B := 298;
	arPM[A5].p_Current_B := 278;
	//arPM[LP_PR1A].p_Current_B := ;
	//arPM[LP_PR1B].p_Current_B := ;
	//arPM[LP_PR2A].p_Current_B := ;
	//arPM[LP_PR2B].p_Current_B := ;
	//arPM[LP_PR3A].p_Current_B := ;
	arPM[DB_WH].p_Current_B := 41.64;
	//arPM[LP_PR3B].p_Current_B := ;
	arPM[LP_PR4A ].p_Current_B := 838;
	arPM[LP_PR4B].p_Current_B := 9.5;
	arPM[LP_BM].p_Current_B :=0.4;
	arPM[DB_BM].p_Current_B := 16.68;
	arPM[LV03].p_Current_B := 1106 ;
	arPM[DB_MVAC1].p_Current_B := 658;
	arPM[DB_MVAC2].p_Current_B :=365;
	arPM[DB_OFF2].p_Current_B := 41 ;
	arPM[LP_EL1].p_Current_B := 0.14;
	arPM[LP_EL2].p_Current_B := 2.5;
	arPM[DB_OFF1].p_Current_B := 62.7;
	arPM[DB_KIT].p_Current_B := 50;
	arPM[LP_WH2].p_Current_B := 45;
	arPM[LP_WH1].p_Current_B := 19.32;
	arPM[CH4].p_Current_B := 0.86;
	arPM[CH5].p_Current_B := 77.4;
	arPM[CH6].p_Current_B := 1.6;
	arPM[LV04].p_Current_B := 602.6;
	arPM[DB_PR2].p_Current_B := 516;
	arPM[DB11].p_Current_B := 19.68;
	arPM[DB12].p_Current_B := 52.6;
	arPM[DB13].p_Current_B := 128.3;
	arPM[DB14].p_Current_B := 171.9;
	arPM[DB11_1].p_Current_B := 27;
	arPM[DB12_1].p_Current_B := 21.16;
	arPM[DB13_1].p_Current_B := 45.97;
	arPM[DB14_1].p_Current_B := 162;
	arPM[DB15].p_Current_B := 212;
	arPM[DB15_1].p_Current_B := 44;
	arPM[LP_PR5A].p_Current_B := 9.18;
	arPM[LP_PR5B].p_Current_B := 9.34;
	arPM[LP_PR6A].p_Current_B := 0.5544;
	arPM[LP_PR6B].p_Current_B := 0.31;
// CurrentC
	arPM[LV01].p_Current_C := 1590;
	arPM[DB_PR1_1].p_Current_C := 1720 ;
	//arPM[DB1].p_Current_C := 50;
	arPM[DB2].p_Current_C :=  58;
	arPM[DB3].p_Current_C := 142;
	arPM[DB4].p_Current_C := 171;
	//arPM[DB1_1].p_Current_C := ;
	arPM[DB2_1].p_Current_C := 25;
	arPM[DB3_1].p_Current_C := 43 ;
	arPM[DB4_1].p_Current_C :=  107;
	//arPM[DB5].p_Current_C := ;
	//arPM[DB6].p_Current_C := ;
	//arPM[DB7].p_Current_C := ;
	arPM[DB_MR].p_Current_C := 2;
	//arPM[DB5_1].p_Current_C := ;
	//arPM[DB6_1].p_Current_C := ;
	//arPM[DB7_1].p_Current_C := ;
	arPM[LV02].p_Current_C := 1650;
	arPM[DB_PR1_2].p_Current_C := 789;
	arPM[DB_AIRCOMP].p_Current_C := 928;
	arPM[DB_AHU].p_Current_C := 149;
	//arPM[DB8].p_Current_C := ;
	//arPM[DB9].p_Current_C := ;
	//arPM[DB10].p_Current_C := ;
	//arPM[DB8_1].p_Current_C := ;
	//arPM[DB9_1].p_Current_C := ;
	//arPM[DB10_1].p_Current_C := ;
	arPM[A1].p_Current_C := 281 ;
	//arPM[A2].p_Current_C := ;
	arPM[A3].p_Current_C := 84 ;
	arPM[A4].p_Current_C := 291;
	arPM[A5].p_Current_C := 246;
	//arPM[LP_PR1A].p_Current_C := ;
	//arPM[LP_PR1B].p_Current_C := ;
	//arPM[LP_PR2A].p_Current_C := ;
	//arPM[LP_PR2B].p_Current_C := ;
	//arPM[LP_PR3A].p_Current_C := ;
	arPM[DB_WH].p_Current_C := 56;
	//arPM[LP_PR3B].p_Current_C := ;
	arPM[LP_PR4A ].p_Current_C := 8.8;
	arPM[LP_PR4B].p_Current_C := 8.5;
	//arPM[LP_BM].p_Current_C := 17.68;
	arPM[DB_BM].p_Current_C := 12.2;
	arPM[LV03].p_Current_C := 1109 ;
	arPM[DB_MVAC1].p_Current_C := 365;
	arPM[DB_MVAC2].p_Current_C :=365;
	arPM[DB_OFF2].p_Current_C := 20 ;
	arPM[LP_EL1].p_Current_C := 1.5;
	arPM[LP_EL2].p_Current_C := 0.4;
	arPM[DB_OFF1].p_Current_C := 70;
	arPM[DB_KIT].p_Current_C := 65;
	arPM[LP_WH2].p_Current_C := 28;
	arPM[LP_WH1].p_Current_C := 21;
	arPM[CH4].p_Current_C := 21;
	arPM[CH5].p_Current_C := 77.4;
	arPM[CH6].p_Current_C := 104;
	arPM[LV04].p_Current_C := 580;
	arPM[DB_PR2].p_Current_C := 544;
	arPM[DB11].p_Current_C := 51;
	arPM[DB12].p_Current_C := 49;
	arPM[DB13].p_Current_C := 75;
	arPM[DB14].p_Current_C := 111;
	arPM[DB11_1].p_Current_C := 4;
	arPM[DB12_1].p_Current_C := 21;
	arPM[DB13_1].p_Current_C := 47.97;
	arPM[DB14_1].p_Current_C := 123;
	arPM[DB15].p_Current_C := 227;
	arPM[DB15_1].p_Current_C := 42;
	arPM[LP_PR5A].p_Current_C := 11.7;
	arPM[LP_PR5B].p_Current_C := 9.6;
	arPM[LP_PR6A].p_Current_C := 0.8;
	arPM[LP_PR6B].p_Current_C := 0.4;
// Real_PowerA 
	arPM[LV01].p_Real_PowerA := 326.48725;
	arPM[DB_PR1_1].p_Real_PowerA := 300.864593505859;
	arPM[DB1].p_Real_PowerA := -88888888.4444;
	arPM[DB2].p_Real_PowerA := 13.6;
	arPM[DB3].p_Real_PowerA := 28.8;
	arPM[DB4].p_Real_PowerA := 41.8;
	arPM[DB1_1].p_Real_PowerA := 0;
	arPM[DB2_1].p_Real_PowerA := 6.16456890106201;
	arPM[DB3_1].p_Real_PowerA := 9.23189353942871;
	arPM[DB4_1].p_Real_PowerA := -1.5E+40;
	arPM[DB5].p_Real_PowerA := -88888888.4444;
	arPM[DB6].p_Real_PowerA := -88888888.4444;
	arPM[DB7].p_Real_PowerA := -88888888.4444;
	arPM[DB_MR].p_Real_PowerA := 4.8;
	arPM[DB5_1].p_Real_PowerA := 0;
	arPM[DB6_1].p_Real_PowerA := 0;
	arPM[DB7_1].p_Real_PowerA := 0;
	arPM[LV02].p_Real_PowerA := 372.88228125;
	arPM[DB_PR1_2].p_Real_PowerA := 135.485427856445;
	arPM[DB_AIRCOMP].p_Real_PowerA := 192.849090576172;
	arPM[DB_AHU].p_Real_PowerA := 32.16;
	arPM[DB8].p_Real_PowerA := -88888888.4444;
	arPM[DB9].p_Real_PowerA := -88888888.4444;
	arPM[DB10].p_Real_PowerA := -88888888.4444;
	arPM[DB8_1].p_Real_PowerA := 0;
	arPM[DB9_1].p_Real_PowerA := 0;
	arPM[DB10_1].p_Real_PowerA := 0;
	arPM[A1].p_Real_PowerA := 58.2002372741699;
	arPM[A2].p_Real_PowerA := 0;
	arPM[A3].p_Real_PowerA := 17.8884391784668;
	arPM[A4].p_Real_PowerA := 59.194408416748;
	arPM[A5].p_Real_PowerA := 50.7736358642578;
	arPM[LP_PR1A].p_Real_PowerA := 0;
	arPM[LP_PR1B].p_Real_PowerA := 0;
	arPM[LP_PR2A].p_Real_PowerA := 0;
	arPM[LP_PR2B].p_Real_PowerA := 0;
	arPM[LP_PR3A].p_Real_PowerA := 0;
	arPM[DB_WH].p_Real_PowerA := 8.16;
	arPM[LP_PR3B].p_Real_PowerA := 0;
	arPM[LP_PR4A ].p_Real_PowerA := 1.92591488361359;
	arPM[LP_PR4B].p_Real_PowerA := 1.82267451286316;
	arPM[LP_BM].p_Real_PowerA := 0.348;
	arPM[DB_BM].p_Real_PowerA := 3.32;
	arPM[LV03].p_Real_PowerA := 232.3538125;
	arPM[DB_MVAC1].p_Real_PowerA := 124.836311340332;
	arPM[DB_MVAC2].p_Real_PowerA := 71.8664169311523;
	arPM[DB_OFF2].p_Real_PowerA := 7860.6;
	arPM[LP_EL1].p_Real_PowerA := 0.928230285644531;
	arPM[LP_EL2].p_Real_PowerA := 0.38;
	arPM[DB_OFF1].p_Real_PowerA := 10.8;
	arPM[DB_KIT].p_Real_PowerA := 10.56;
	arPM[LP_WH2].p_Real_PowerA := 7.57289457321167;
	arPM[LP_WH1].p_Real_PowerA := 4.67977142333984;
	arPM[CH4].p_Real_PowerA := 13.279465675354;
	arPM[CH5].p_Real_PowerA := 0.173617959022522;
	arPM[CH6].p_Real_PowerA := 20.3546371459961;
	arPM[LV04].p_Real_PowerA := 121.57978125;
	arPM[DB_PR2].p_Real_PowerA := 114.4;
	arPM[DB11].p_Real_PowerA := 10.72;
	arPM[DB12].p_Real_PowerA := 9.3;
	arPM[DB13].p_Real_PowerA := 20.48;
	arPM[DB14].p_Real_PowerA := 36.16;
	arPM[DB11_1].p_Real_PowerA := 6.06992387771606;
	arPM[DB12_1].p_Real_PowerA := 4.43687963485718;
	arPM[DB13_1].p_Real_PowerA := 10.6720571517944;
	arPM[DB14_1].p_Real_PowerA := 31.2415618896484;
	arPM[DB15].p_Real_PowerA := 37.12;
	arPM[DB15_1].p_Real_PowerA := 7.1462984085083;
	arPM[LP_PR5A].p_Real_PowerA := -2.05480074882507;
	arPM[LP_PR5B].p_Real_PowerA := 1.89803433418274;
	arPM[LP_PR6A].p_Real_PowerA := 0.0984331741929054;
	arPM[LP_PR6B].p_Real_PowerA := 0.0509700253605843;
	
// p_Real_PowerB
	arPM[LV01].p_Real_PowerB := 350.48725;
	arPM[DB_PR1_1].p_Real_PowerB := 320.864593505859;
	arPM[DB1].p_Real_PowerB := -88888888.4444;
	arPM[DB2].p_Real_PowerB := 12.24;
	arPM[DB3].p_Real_PowerB := 35.28;
	arPM[DB4].p_Real_PowerB := 43.4;
	arPM[DB1_1].p_Real_PowerB := 0;
	arPM[DB2_1].p_Real_PowerB := 11.4156036376953;
	arPM[DB3_1].p_Real_PowerB := -1.5E+40;
	arPM[DB4_1].p_Real_PowerB := 15.1349725723267;
	arPM[DB5].p_Real_PowerB := -88888888.4444;
	arPM[DB6].p_Real_PowerB := -88888888.4444;
	arPM[DB7].p_Real_PowerB := -88888888.4444;
	arPM[DB_MR].p_Real_PowerB := 9.06;
	arPM[DB5_1].p_Real_PowerB := 0;
	arPM[DB6_1].p_Real_PowerB := 0;
	arPM[DB7_1].p_Real_PowerB := 0;
	arPM[LV02].p_Real_PowerB := 384.8741875;
	arPM[DB_PR1_2].p_Real_PowerB := 152.953918457031;
	arPM[DB_AIRCOMP].p_Real_PowerB := 199.420104980469;
	arPM[DB_AHU].p_Real_PowerB := 32.76;
	arPM[DB8].p_Real_PowerB := -88888888.4444;
	arPM[DB9].p_Real_PowerB := -88888888.4444;
	arPM[DB10].p_Real_PowerB := -88888888.4444;
	arPM[DB8_1].p_Real_PowerB := 0;
	arPM[DB9_1].p_Real_PowerB := 0;
	arPM[DB10_1].p_Real_PowerB := 0;
	arPM[A1].p_Real_PowerB := 59.1645774841309;
	arPM[A2].p_Real_PowerB := 0;
	arPM[A3].p_Real_PowerB := 20.5810832977295;
	arPM[A4].p_Real_PowerB := -1.5E+40;
	arPM[A5].p_Real_PowerB := -1.5E+40;
	arPM[LP_PR1A].p_Real_PowerB := 0;
	arPM[LP_PR1B].p_Real_PowerB := 0;
	arPM[LP_PR2A].p_Real_PowerB := 0;
	arPM[LP_PR2B].p_Real_PowerB := 0;
	arPM[LP_PR3A].p_Real_PowerB := 0;
	arPM[DB_WH].p_Real_PowerB := 5.88;
	arPM[LP_PR3B].p_Real_PowerB := 0;
	arPM[LP_PR4A ].p_Real_PowerB := -1.5E+40;
	arPM[LP_PR4B].p_Real_PowerB := -1.5E+40;
	arPM[LP_BM].p_Real_PowerB := 0.048;
	arPM[DB_BM].p_Real_PowerB := 0.52;
	arPM[LV03].p_Real_PowerB := 242.520046875;
	arPM[DB_MVAC1].p_Real_PowerB := 124.868919372559;
	arPM[DB_MVAC2].p_Real_PowerB := 77.7159729003906;
	arPM[DB_OFF2].p_Real_PowerB := 6.6;
	arPM[LP_EL1].p_Real_PowerB := 0.0135234519839287;
	arPM[LP_EL2].p_Real_PowerB := 0.16;
	arPM[DB_OFF1].p_Real_PowerB := 11.5;
	arPM[DB_KIT].p_Real_PowerB := 14.88;
	arPM[LP_WH2].p_Real_PowerB := 10.351185798645;
	arPM[LP_WH1].p_Real_PowerB := 5.06796789169312;
	arPM[CH4].p_Real_PowerB := 13.4788665771484;
	arPM[CH5].p_Real_PowerB := 0.132516324520111;
	arPM[CH6].p_Real_PowerB := 20.9350357055664;
	arPM[LV04].p_Real_PowerB := 113.8976640625;
	arPM[DB_PR2].p_Real_PowerB := 141.6;
	arPM[DB11].p_Real_PowerB := 8.88;
	arPM[DB12].p_Real_PowerB := 7.6;
	arPM[DB13].p_Real_PowerB := 21.12;
	arPM[DB14].p_Real_PowerB := 29.12;
	arPM[DB11_1].p_Real_PowerB := 4.97021770477295;
	arPM[DB12_1].p_Real_PowerB := 4.62906122207642;
	arPM[DB13_1].p_Real_PowerB := 9.47135925292969;
	arPM[DB14_1].p_Real_PowerB := 21.6200199127197;
	arPM[DB15].p_Real_PowerB := 38.72;
	arPM[DB15_1].p_Real_PowerB := 8.88123321533203;
	arPM[LP_PR5A].p_Real_PowerB := 1.63270902633667;
	arPM[LP_PR5B].p_Real_PowerB := 1.82756507396698;
	arPM[LP_PR6A].p_Real_PowerB := 0.0718437507748604;
	arPM[LP_PR6B].p_Real_PowerB := 0.0553829297423363;
// p_Real_PowerC
	arPM[LV01].p_Real_PowerC := 281.90271875;
	arPM[DB_PR1_1].p_Real_PowerC := 295.549530029297;
	arPM[DB1].p_Real_PowerC := -88888888.4444;
	arPM[DB2].p_Real_PowerC := 11.68;
	arPM[DB3].p_Real_PowerC := 33.84;
	arPM[DB4].p_Real_PowerC := 2.2;
	arPM[DB1_1].p_Real_PowerC := 0;
	arPM[DB2_1].p_Real_PowerC := -1.5E+40;
	arPM[DB3_1].p_Real_PowerC := 7.25864553451538;
	arPM[DB4_1].p_Real_PowerC := 14.5833835601807;
	arPM[DB5].p_Real_PowerC := -88888888.4444;
	arPM[DB6].p_Real_PowerC := -88888888.4444;
	arPM[DB7].p_Real_PowerC := -88888888.4444;
	arPM[DB_MR].p_Real_PowerC := 5.7;
	arPM[DB5_1].p_Real_PowerC := 0;
	arPM[DB6_1].p_Real_PowerC := 0;
	arPM[DB7_1].p_Real_PowerC := 0;
	arPM[LV02].p_Real_PowerC := 370.28871875;
	arPM[DB_PR1_2].p_Real_PowerC := 145.278213500977;
	arPM[DB_AIRCOMP].p_Real_PowerC := 195.644317626953;
	arPM[DB_AHU].p_Real_PowerC := 32.04;
	arPM[DB8].p_Real_PowerC := -88888888.4444;
	arPM[DB9].p_Real_PowerC := -88888888.4444;
	arPM[DB10].p_Real_PowerC := -88888888.4444;
	arPM[DB8_1].p_Real_PowerC := 0;
	arPM[DB9_1].p_Real_PowerC := 0;
	arPM[DB10_1].p_Real_PowerC := 0;
	arPM[A1].p_Real_PowerC := -1.5E+40;
	arPM[A2].p_Real_PowerC := 0;
	arPM[A3].p_Real_PowerC := 16.4717750549316;
	arPM[A4].p_Real_PowerC := 58.0558242797852;
	arPM[A5].p_Real_PowerC := 44.6190452575684;
	arPM[LP_PR1A].p_Real_PowerC := 0;
	arPM[LP_PR1B].p_Real_PowerC := 0;
	arPM[LP_PR2A].p_Real_PowerC := 0;
	arPM[LP_PR2B].p_Real_PowerC := 0;
	arPM[LP_PR3A].p_Real_PowerC := 0;
	arPM[DB_WH].p_Real_PowerC := 5.16;
	arPM[LP_PR3B].p_Real_PowerC := 0;
	arPM[LP_PR4A ].p_Real_PowerC := -1.5E+40;
	arPM[LP_PR4B].p_Real_PowerC := -1.5E+40;
	arPM[LP_BM].p_Real_PowerC := 0;
	arPM[DB_BM].p_Real_PowerC := 0.88;
	arPM[LV03].p_Real_PowerC := 237.472578125;
	arPM[DB_MVAC1].p_Real_PowerC := -1.5E+40;
	arPM[DB_MVAC2].p_Real_PowerC := 73.6659088134766;
	arPM[DB_OFF2].p_Real_PowerC := 7.08;
	arPM[LP_EL1].p_Real_PowerC := 0.249511554837227;
	arPM[LP_EL2].p_Real_PowerC := 0.06;
	arPM[DB_OFF1].p_Real_PowerC := 11.3;
	arPM[DB_KIT].p_Real_PowerC := 10.64;
	arPM[LP_WH2].p_Real_PowerC := 5.57862091064453;
	arPM[LP_WH1].p_Real_PowerC := 4.88177013397217;
	arPM[CH4].p_Real_PowerC := 12.4203805923462;
	arPM[CH5].p_Real_PowerC := 0;
	arPM[CH6].p_Real_PowerC := 19.1779308319092;
	arPM[LV04].p_Real_PowerC := 107.71028125;
	arPM[DB_PR2].p_Real_PowerC := 128.8;
	arPM[DB11].p_Real_PowerC := 12.16;
	arPM[DB12].p_Real_PowerC := 7.9;
	arPM[DB13].p_Real_PowerC := 14.72;
	arPM[DB14].p_Real_PowerC := 21.76;
	arPM[DB11_1].p_Real_PowerC := 2.55743432044983;
	arPM[DB12_1].p_Real_PowerC := 4.93209791183472;
	arPM[DB13_1].p_Real_PowerC := 8.78751564025879;
	arPM[DB14_1].p_Real_PowerC := 24.1240062713623;
	arPM[DB15].p_Real_PowerC := 51.52;
	arPM[DB15_1].p_Real_PowerC := 8.43356513977051;
	arPM[LP_PR5A].p_Real_PowerC := 2.17041778564453;
	arPM[LP_PR5B].p_Real_PowerC := 2.04661750793457;
	arPM[LP_PR6A].p_Real_PowerC := 0.15382182598114;
	arPM[LP_PR6B].p_Real_PowerC := 0.0687989294528961;
//	p_RealEnergy_IntoLoad
	arPM[LV01].p_RealEnergy_IntoLoad := LV01_Real_RealEnergy_IntoLoad;
	arPM[DB_PR1_1].p_RealEnergy_IntoLoad := DB_PR1_1_Real_RealEnergy_IntoLoad;
	arPM[DB1].p_RealEnergy_IntoLoad := DB1_Real_RealEnergy_IntoLoad;
	arPM[DB2].p_RealEnergy_IntoLoad := DB2_Real_RealEnergy_IntoLoad;
	arPM[DB3].p_RealEnergy_IntoLoad := DB3_Real_RealEnergy_IntoLoad;
	arPM[DB4].p_RealEnergy_IntoLoad := DB4_Real_RealEnergy_IntoLoad;
	arPM[DB1_1].p_RealEnergy_IntoLoad := DB1_1_Real_RealEnergy_IntoLoad;
	arPM[DB2_1].p_RealEnergy_IntoLoad := DB2_1_Real_RealEnergy_IntoLoad;
	arPM[DB3_1].p_RealEnergy_IntoLoad := DB3_1_Real_RealEnergy_IntoLoad;
	arPM[DB4_1].p_RealEnergy_IntoLoad := DB4_1_Real_RealEnergy_IntoLoad;
	arPM[DB5].p_RealEnergy_IntoLoad := DB5_Real_RealEnergy_IntoLoad;
	arPM[DB6].p_RealEnergy_IntoLoad := DB6_Real_RealEnergy_IntoLoad;
	arPM[DB7].p_RealEnergy_IntoLoad := DB7_Real_RealEnergy_IntoLoad;
	arPM[DB_MR].p_RealEnergy_IntoLoad := DB_MR_Real_RealEnergy_IntoLoad;
	arPM[DB5_1].p_RealEnergy_IntoLoad := DB5_1_Real_RealEnergy_IntoLoad;
	arPM[DB6_1].p_RealEnergy_IntoLoad := DB6_1_Real_RealEnergy_IntoLoad;
	arPM[DB7_1].p_RealEnergy_IntoLoad := DB7_1_Real_RealEnergy_IntoLoad;
	arPM[LV02].p_RealEnergy_IntoLoad := LV02_Real_RealEnergy_IntoLoad;
	arPM[DB_PR1_2].p_RealEnergy_IntoLoad := DB_PR1_2_Real_RealEnergy_IntoLoad;
	arPM[DB_AIRCOMP].p_RealEnergy_IntoLoad := DB_AIRCOMP_Real_RealEnergy_IntoLoad;
	arPM[DB_AHU].p_RealEnergy_IntoLoad := DB_AHU_Real_RealEnergy_IntoLoad;
	arPM[DB8].p_RealEnergy_IntoLoad := DB8_Real_RealEnergy_IntoLoad;
	arPM[DB9].p_RealEnergy_IntoLoad := DB9_Real_RealEnergy_IntoLoad;
	arPM[DB10].p_RealEnergy_IntoLoad := DB10_Real_RealEnergy_IntoLoad;
	arPM[DB8_1].p_RealEnergy_IntoLoad := DB8_1_Real_RealEnergy_IntoLoad;
	arPM[DB9_1].p_RealEnergy_IntoLoad := DB9_1_Real_RealEnergy_IntoLoad;
	arPM[DB10_1].p_RealEnergy_IntoLoad := DB10_1_Real_RealEnergy_IntoLoad;
	arPM[A1].p_RealEnergy_IntoLoad := A1_Real_RealEnergy_IntoLoad;
	arPM[A2].p_RealEnergy_IntoLoad := A2_Real_RealEnergy_IntoLoad;
	arPM[A3].p_RealEnergy_IntoLoad := A3_Real_RealEnergy_IntoLoad;
	arPM[A4].p_RealEnergy_IntoLoad := A4_Real_RealEnergy_IntoLoad;
	arPM[A5].p_RealEnergy_IntoLoad := A5_Real_RealEnergy_IntoLoad;
	arPM[LP_PR1A].p_RealEnergy_IntoLoad := LP_PR1A_Real_RealEnergy_IntoLoad;
	arPM[LP_PR1B].p_RealEnergy_IntoLoad := LP_PR1B_Real_RealEnergy_IntoLoad;
	arPM[LP_PR2A].p_RealEnergy_IntoLoad := LP_PR2A_Real_RealEnergy_IntoLoad;
	arPM[LP_PR2B].p_RealEnergy_IntoLoad := LP_PR2B_Real_RealEnergy_IntoLoad;
	arPM[LP_PR3A].p_RealEnergy_IntoLoad := LP_PR3A_Real_RealEnergy_IntoLoad;
	arPM[DB_WH].p_RealEnergy_IntoLoad := DB_WH_Real_RealEnergy_IntoLoad;
	arPM[LP_PR3B].p_RealEnergy_IntoLoad := LP_PR3B_Real_RealEnergy_IntoLoad;
	arPM[LP_PR4A].p_RealEnergy_IntoLoad := LP_PR4A_Real_RealEnergy_IntoLoad;
	arPM[LP_PR4B].p_RealEnergy_IntoLoad := LP_PR4B_Real_RealEnergy_IntoLoad;
	arPM[LP_BM].p_RealEnergy_IntoLoad := LP_BM_Real_RealEnergy_IntoLoad;
	arPM[DB_BM].p_RealEnergy_IntoLoad := DB_BM_Real_RealEnergy_IntoLoad;
	arPM[LV03].p_RealEnergy_IntoLoad := LV03_Real_RealEnergy_IntoLoad;
	arPM[DB_MVAC1].p_RealEnergy_IntoLoad := DB_MVAC1_Real_RealEnergy_IntoLoad;
	arPM[DB_MVAC2].p_RealEnergy_IntoLoad := DB_MVAC2_Real_RealEnergy_IntoLoad;
	arPM[DB_OFF2].p_RealEnergy_IntoLoad := DB_OFF2_Real_RealEnergy_IntoLoad;
	arPM[LP_EL1].p_RealEnergy_IntoLoad := LP_EL1_Real_RealEnergy_IntoLoad;
	arPM[LP_EL2].p_RealEnergy_IntoLoad := LP_EL2_Real_RealEnergy_IntoLoad;
	arPM[DB_OFF1].p_RealEnergy_IntoLoad := DB_OFF1_Real_RealEnergy_IntoLoad;
	arPM[DB_KIT].p_RealEnergy_IntoLoad := DB_KIT_Real_RealEnergy_IntoLoad;
	arPM[LP_WH2].p_RealEnergy_IntoLoad := LP_WH2_Real_RealEnergy_IntoLoad;
	arPM[LP_WH1].p_RealEnergy_IntoLoad := LP_WH1_Real_RealEnergy_IntoLoad;
	arPM[CH4].p_RealEnergy_IntoLoad := CH4_Real_RealEnergy_IntoLoad;
	arPM[CH5].p_RealEnergy_IntoLoad := CH5_Real_RealEnergy_IntoLoad;
	arPM[CH6].p_RealEnergy_IntoLoad := CH6_Real_RealEnergy_IntoLoad;
	arPM[LV04].p_RealEnergy_IntoLoad := LV04_Real_RealEnergy_IntoLoad;
	arPM[DB_PR2].p_RealEnergy_IntoLoad := DB_PR2_Real_RealEnergy_IntoLoad;
	arPM[DB11].p_RealEnergy_IntoLoad := DB11_Real_RealEnergy_IntoLoad;
	arPM[DB12].p_RealEnergy_IntoLoad := DB12_Real_RealEnergy_IntoLoad;
	arPM[DB13].p_RealEnergy_IntoLoad := DB13_Real_RealEnergy_IntoLoad;
	arPM[DB14].p_RealEnergy_IntoLoad := DB14_Real_RealEnergy_IntoLoad;
	arPM[DB11_1].p_RealEnergy_IntoLoad := DB11_1_Real_RealEnergy_IntoLoad;
	arPM[DB12_1].p_RealEnergy_IntoLoad := DB12_1_Real_RealEnergy_IntoLoad;
	arPM[DB13_1].p_RealEnergy_IntoLoad := DB13_1_Real_RealEnergy_IntoLoad;
	arPM[DB14_1].p_RealEnergy_IntoLoad := DB14_1_Real_RealEnergy_IntoLoad;
	arPM[DB15].p_RealEnergy_IntoLoad := DB15_Real_RealEnergy_IntoLoad;
	arPM[DB15_1].p_RealEnergy_IntoLoad := DB15_1_Real_RealEnergy_IntoLoad;
	arPM[LP_PR5A].p_RealEnergy_IntoLoad := LP_PR5A_Real_RealEnergy_IntoLoad;
	arPM[LP_PR5B].p_RealEnergy_IntoLoad := LP_PR5B_Real_RealEnergy_IntoLoad;
	arPM[LP_PR6A].p_RealEnergy_IntoLoad := LP_PR6A_Real_RealEnergy_IntoLoad;
	arPM[LP_PR6B].p_RealEnergy_IntoLoad := LP_PR6B_Real_RealEnergy_IntoLoad;
	
// update dentalRealEnergy_IntoLoad
	arPM[LV01].p_dentalRealEnergy_IntoLoad := 81.4864739239071;
	arPM[DB_PR1_1].p_dentalRealEnergy_IntoLoad := 80.361624988331;
	arPM[DB1].p_dentalRealEnergy_IntoLoad := 0;
	arPM[DB2].p_dentalRealEnergy_IntoLoad := 3.43962071209237;
	arPM[DB3].p_dentalRealEnergy_IntoLoad := 7.61364692757743;
	arPM[DB4].p_dentalRealEnergy_IntoLoad := 7.02333364320482;
	arPM[DB1_1].p_dentalRealEnergy_IntoLoad := 0;
	arPM[DB2_1].p_dentalRealEnergy_IntoLoad := 1.16203402435553;
	arPM[DB3_1].p_dentalRealEnergy_IntoLoad := 1.98010597750182;
	arPM[DB4_1].p_dentalRealEnergy_IntoLoad := 3.70456446964543;
	arPM[DB5].p_dentalRealEnergy_IntoLoad := 0;
	arPM[DB6].p_dentalRealEnergy_IntoLoad := 0;
	arPM[DB7].p_dentalRealEnergy_IntoLoad := 0;
	arPM[DB_MR].p_dentalRealEnergy_IntoLoad := 0.599609556567453;
	arPM[DB5_1].p_dentalRealEnergy_IntoLoad := 0;
	arPM[DB6_1].p_dentalRealEnergy_IntoLoad := 0;
	arPM[DB7_1].p_dentalRealEnergy_IntoLoad := 0;
	arPM[LV02].p_dentalRealEnergy_IntoLoad := 96.1931765361507;
	arPM[DB_PR1_2].p_dentalRealEnergy_IntoLoad := 39.2256205261452;
	arPM[DB_AIRCOMP].p_dentalRealEnergy_IntoLoad := 48.2615970995338;
	arPM[DB_AHU].p_dentalRealEnergy_IntoLoad := 8.1342381704887;
	arPM[DB8].p_dentalRealEnergy_IntoLoad := 0;
	arPM[DB9].p_dentalRealEnergy_IntoLoad := 0;
	arPM[DB10].p_dentalRealEnergy_IntoLoad := 0;
	arPM[DB8_1].p_dentalRealEnergy_IntoLoad := 0;
	arPM[DB9_1].p_dentalRealEnergy_IntoLoad := 0;
	arPM[DB10_1].p_dentalRealEnergy_IntoLoad := 0;
	arPM[A1].p_dentalRealEnergy_IntoLoad := 14.678813795659;
	arPM[A2].p_dentalRealEnergy_IntoLoad := 0;
	arPM[A3].p_dentalRealEnergy_IntoLoad := 5.05717207399526;
	arPM[A4].p_dentalRealEnergy_IntoLoad := 14.8229060146791;
	arPM[A5].p_dentalRealEnergy_IntoLoad := 11.550618202094;
	arPM[LP_PR1A].p_dentalRealEnergy_IntoLoad := 0;
	arPM[LP_PR1B].p_dentalRealEnergy_IntoLoad := 0;
	arPM[LP_PR2A].p_dentalRealEnergy_IntoLoad := 0;
	arPM[LP_PR2B].p_dentalRealEnergy_IntoLoad := 0;
	arPM[LP_PR3A].p_dentalRealEnergy_IntoLoad := 0;
	arPM[DB_WH].p_dentalRealEnergy_IntoLoad := 1.58036627312352;
	arPM[LP_PR3B].p_dentalRealEnergy_IntoLoad := 0;
	arPM[LP_PR4A].p_dentalRealEnergy_IntoLoad := 0.460165473644789;
	arPM[LP_PR4B].p_dentalRealEnergy_IntoLoad := 0.469461745839634;
	arPM[LP_BM].p_dentalRealEnergy_IntoLoad := 0.0511294970716433;
	arPM[DB_BM].p_dentalRealEnergy_IntoLoad := 0.57172073998292;
	arPM[LV03].p_dentalRealEnergy_IntoLoad := 60.4118248581952;
	arPM[DB_MVAC1].p_dentalRealEnergy_IntoLoad := 30.0594961420288;
	arPM[DB_MVAC2].p_dentalRealEnergy_IntoLoad := 18.4763409872529;
	arPM[DB_OFF2].p_dentalRealEnergy_IntoLoad := 2.66338198382287;
	arPM[LP_EL1].p_dentalRealEnergy_IntoLoad := 0.515943106813855;
	arPM[LP_EL2].p_dentalRealEnergy_IntoLoad := 0.260295621455638;
	arPM[DB_OFF1].p_dentalRealEnergy_IntoLoad := 2.56577112577701;
	arPM[DB_KIT].p_dentalRealEnergy_IntoLoad := 1.849958166774;
	arPM[LP_WH2].p_dentalRealEnergy_IntoLoad := 2.35195686529559;
	arPM[LP_WH1].p_dentalRealEnergy_IntoLoad := 1.20386724923233;
	arPM[CH4].p_dentalRealEnergy_IntoLoad := 1.7662917170204;
	arPM[CH5].p_dentalRealEnergy_IntoLoad := 1.56177372873383;
	arPM[CH6].p_dentalRealEnergy_IntoLoad := 5.14083852374886;
	arPM[LV04].p_dentalRealEnergy_IntoLoad := 31.3144928883328;
	arPM[DB_PR2].p_dentalRealEnergy_IntoLoad := 31.0449009946823;
	arPM[DB11].p_dentalRealEnergy_IntoLoad := 2.16138328530128;
	arPM[DB12].p_dentalRealEnergy_IntoLoad := 2.62154875894607;
	arPM[DB13].p_dentalRealEnergy_IntoLoad := 4.88054290229322;
	arPM[DB14].p_dentalRealEnergy_IntoLoad := 8.05521985683253;
	arPM[DB11_1].p_dentalRealEnergy_IntoLoad := 0.492702426326744;
	arPM[DB12_1].p_dentalRealEnergy_IntoLoad := 0.952867899971534;
	arPM[DB13_1].p_dentalRealEnergy_IntoLoad := 2.31012364041879;
	arPM[DB14_1].p_dentalRealEnergy_IntoLoad := 7.18601840661459;
	arPM[DB15].p_dentalRealEnergy_IntoLoad := 11.6575253323347;
	arPM[DB15_1].p_dentalRealEnergy_IntoLoad := 1.99869852189151;
	arPM[LP_PR5A].p_dentalRealEnergy_IntoLoad := 0.134795946825241;
	arPM[LP_PR5B].p_dentalRealEnergy_IntoLoad := 0.488054290229322;
	arPM[LP_PR6A].p_dentalRealEnergy_IntoLoad := 0.0278888165845327;
	arPM[LP_PR6B].p_dentalRealEnergy_IntoLoad := 0.0139444082922663;


// p_RealEnergy_OutLoad
	arPM[LV01].p_ReactiveEnergy_OutLoad := 6873.314;
	arPM[DB_PR1_1].p_ReactiveEnergy_OutLoad := 7541.118;
	arPM[DB1].p_ReactiveEnergy_OutLoad := -88888888.4444;
	arPM[DB2].p_ReactiveEnergy_OutLoad := -88888888.4444;
	arPM[DB3].p_ReactiveEnergy_OutLoad := -88888888.4444;
	arPM[DB4].p_ReactiveEnergy_OutLoad := -88888888.4444;
	arPM[DB1_1].p_ReactiveEnergy_OutLoad := -88888888.4444;
	arPM[DB2_1].p_ReactiveEnergy_OutLoad := 0;
	arPM[DB3_1].p_ReactiveEnergy_OutLoad := -88888888.4444;
	arPM[DB4_1].p_ReactiveEnergy_OutLoad := 182030.718;
	arPM[DB5].p_ReactiveEnergy_OutLoad := -88888888.4444;
	arPM[DB6].p_ReactiveEnergy_OutLoad := -0.001;
	arPM[DB7].p_ReactiveEnergy_OutLoad := -88888888.4444;
	arPM[DB_MR].p_ReactiveEnergy_OutLoad := -0.001;
	arPM[DB5_1].p_ReactiveEnergy_OutLoad := -88888888.4444;
	arPM[DB6_1].p_ReactiveEnergy_OutLoad := -88888888.4444;
	arPM[DB7_1].p_ReactiveEnergy_OutLoad := -88888888.4444;
	arPM[LV02].p_ReactiveEnergy_OutLoad := -88888888.4444;
	arPM[DB_PR1_2].p_ReactiveEnergy_OutLoad := -88888888.4444;
	arPM[DB_AIRCOMP].p_ReactiveEnergy_OutLoad := 0;
	arPM[DB_AHU].p_ReactiveEnergy_OutLoad := -88888888.4444;
	arPM[DB8].p_ReactiveEnergy_OutLoad := 0;
	arPM[DB9].p_ReactiveEnergy_OutLoad := -88888888.4444;
	arPM[DB10].p_ReactiveEnergy_OutLoad := 0;
	arPM[DB8_1].p_ReactiveEnergy_OutLoad := 9729.96;
	arPM[DB9_1].p_ReactiveEnergy_OutLoad := 11119.27;
	arPM[DB10_1].p_ReactiveEnergy_OutLoad := 24.853;
	arPM[A1].p_ReactiveEnergy_OutLoad := -88888888.4444;
	arPM[A2].p_ReactiveEnergy_OutLoad := -88888888.4444;
	arPM[A3].p_ReactiveEnergy_OutLoad := -88888888.4444;
	arPM[A4].p_ReactiveEnergy_OutLoad := -88888888.4444;
	arPM[A5].p_ReactiveEnergy_OutLoad := -88888888.4444;
	arPM[LP_PR1A].p_ReactiveEnergy_OutLoad := 0;
	arPM[LP_PR1B].p_ReactiveEnergy_OutLoad := -88888888.4444;
	arPM[LP_PR2A].p_ReactiveEnergy_OutLoad := 0;
	arPM[LP_PR2B].p_ReactiveEnergy_OutLoad := -88888888.4444;
	arPM[LP_PR3A].p_ReactiveEnergy_OutLoad := 0;
	arPM[DB_WH].p_ReactiveEnergy_OutLoad := 0;
	arPM[LP_PR3B].p_ReactiveEnergy_OutLoad := 0;
	arPM[LP_PR4A ].p_ReactiveEnergy_OutLoad := -0.001;
	arPM[LP_PR4B].p_ReactiveEnergy_OutLoad := -0.001;
	arPM[LP_BM].p_ReactiveEnergy_OutLoad := 206.65;
	arPM[DB_BM].p_ReactiveEnergy_OutLoad := 0;
	arPM[LV03].p_ReactiveEnergy_OutLoad := 0;
	arPM[DB_MVAC1].p_ReactiveEnergy_OutLoad := 0;
	arPM[DB_MVAC2].p_ReactiveEnergy_OutLoad := 0;
	arPM[DB_OFF2].p_ReactiveEnergy_OutLoad := 0;
	arPM[LP_EL1].p_ReactiveEnergy_OutLoad := -88888888.4444;
	arPM[LP_EL2].p_ReactiveEnergy_OutLoad := 0;
	arPM[DB_OFF1].p_ReactiveEnergy_OutLoad := 212932.137;
	arPM[DB_KIT].p_ReactiveEnergy_OutLoad := 216938.692;
	arPM[LP_WH2].p_ReactiveEnergy_OutLoad := -88888888.4444;
	arPM[LP_WH1].p_ReactiveEnergy_OutLoad := -88888888.4444;
	arPM[CH4].p_ReactiveEnergy_OutLoad := 25920.378;
	arPM[CH5].p_ReactiveEnergy_OutLoad := 27.906;
	arPM[CH6].p_ReactiveEnergy_OutLoad := 785.01;
	arPM[LV04].p_ReactiveEnergy_OutLoad := -88888888.4444;
	arPM[DB_PR2].p_ReactiveEnergy_OutLoad := 32352.822;
	arPM[DB11].p_ReactiveEnergy_OutLoad := -88888888.4444;
	arPM[DB12].p_ReactiveEnergy_OutLoad := -88888888.4444;
	arPM[DB13].p_ReactiveEnergy_OutLoad := -88888888.4444;
	arPM[DB14].p_ReactiveEnergy_OutLoad := 7123.4;
	arPM[DB11_1].p_ReactiveEnergy_OutLoad := 11321.767;
	arPM[DB12_1].p_ReactiveEnergy_OutLoad := 0.004;
	arPM[DB13_1].p_ReactiveEnergy_OutLoad := 0;
	arPM[DB14_1].p_ReactiveEnergy_OutLoad := 0;
	arPM[DB15].p_ReactiveEnergy_OutLoad := 4383.502;
	arPM[DB15_1].p_ReactiveEnergy_OutLoad := -88888888.4444;
	arPM[LP_PR5A].p_ReactiveEnergy_OutLoad := -88888888.4444;
	arPM[LP_PR5B].p_ReactiveEnergy_OutLoad := -88888888.4444;
	arPM[LP_PR6A].p_ReactiveEnergy_OutLoad := -88888888.4444;
	arPM[LP_PR6B].p_ReactiveEnergy_OutLoad := -88888888.4444;

